// SIMATIC S7-200 SMART project (STEP 7-Micro/WIN SMART), CPU ST20

SYMBOL_TABLE System Symbols
Always_On        SM0.0    // Always ON
First_Scan_On    SM0.1    // ON for the first scan cycle only
Clock_1s         SM0.5    // Clock pulse that is ON for 0.5 s, OFF for 0.5 s, for a duty cycle time of 1 s.
END_SYMBOL_TABLE

SYMBOL_TABLE Modbus RTU Master2 (v2.0)
mModbusBufrFctn  VB420    // Modbusbufr[2] - function code byte
END_SYMBOL_TABLE

ORGANIZATION_BLOCK MAIN:OB1
TITLE=Program Comments
BEGIN
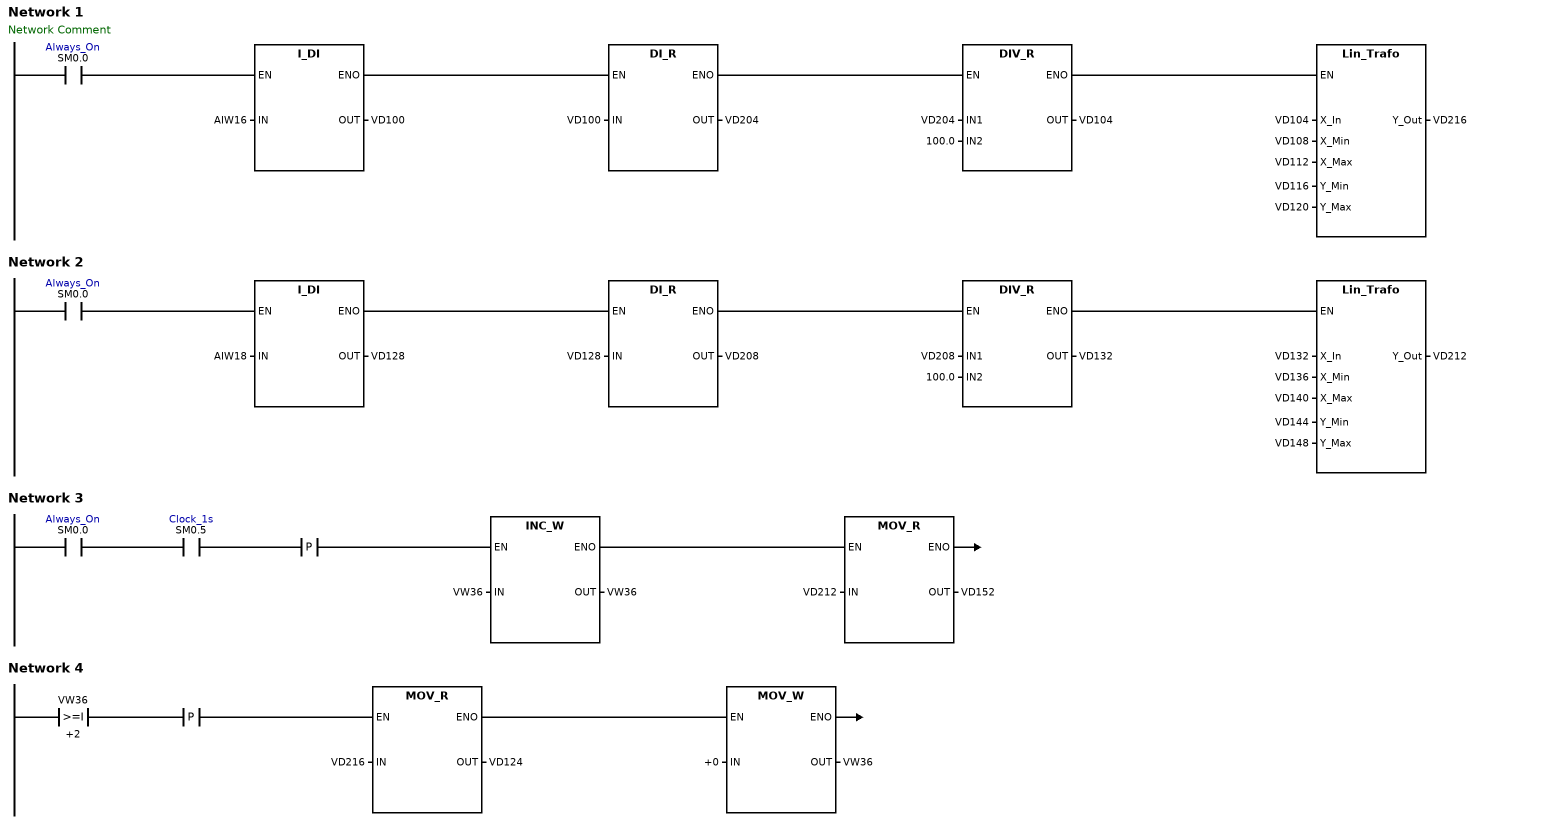
Network 1
// Network Comment
LD     Always_On:SM0.0
ITD    AIW16, VD100
AENO
DTR    VD100, VD204
AENO
MOVR   VD204, VD104
AENO
/R     100.0, VD104
AENO
CALL   Lin_Trafo:SBR1, VD104, VD108, VD112, VD116, VD120, VD216
Network 2
LD     Always_On:SM0.0
ITD    AIW18, VD128
AENO
DTR    VD128, VD208
AENO
MOVR   VD208, VD132
AENO
/R     100.0, VD132
AENO
CALL   Lin_Trafo:SBR1, VD132, VD136, VD140, VD144, VD148, VD212
Network 3
LD     Always_On:SM0.0
A      Clock_1s:SM0.5
EU
INCW   VW36
AENO
MOVR   VD212, VD152
Network 4
LDW>=  VW36, +2
EU
MOVR   VD216, VD124
AENO
MOVW   +0, VW36
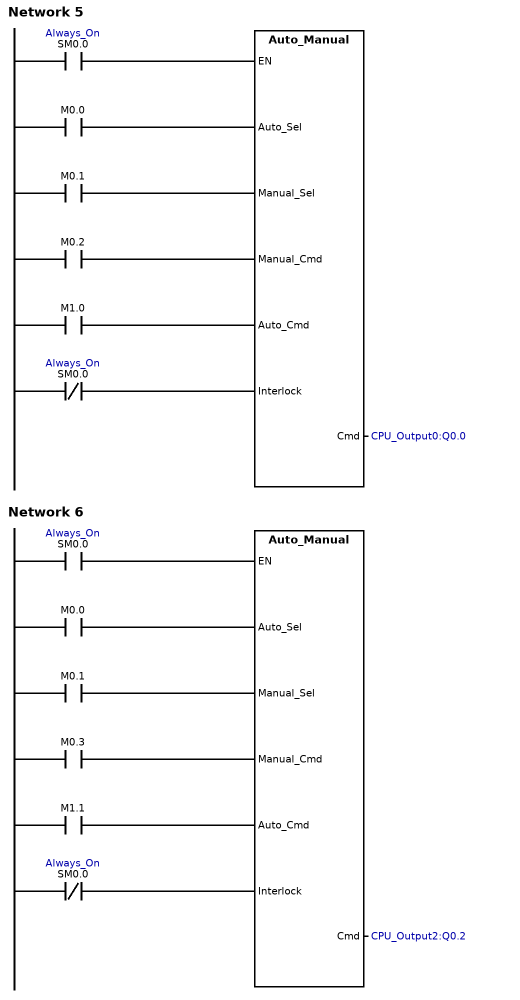
Network 5
LD     Always_On:SM0.0
=      L60.0
LD     M0.0
=      L63.7
LD     M0.1
=      L63.6
LD     M0.2
=      L63.5
LD     M1.0
=      L63.4
LDN    Always_On:SM0.0
=      L63.3
LD     L60.0
CALL   Auto_Manual:SBR2, L63.7, L63.6, L63.5, L63.4, L63.3, CPU_Output0:Q0.0
Network 6
LD     Always_On:SM0.0
=      L60.0
LD     M0.0
=      L63.7
LD     M0.1
=      L63.6
LD     M0.3
=      L63.5
LD     M1.1
=      L63.4
LDN    Always_On:SM0.0
=      L63.3
LD     L60.0
CALL   Auto_Manual:SBR2, L63.7, L63.6, L63.5, L63.4, L63.3, CPU_Output2:Q0.2
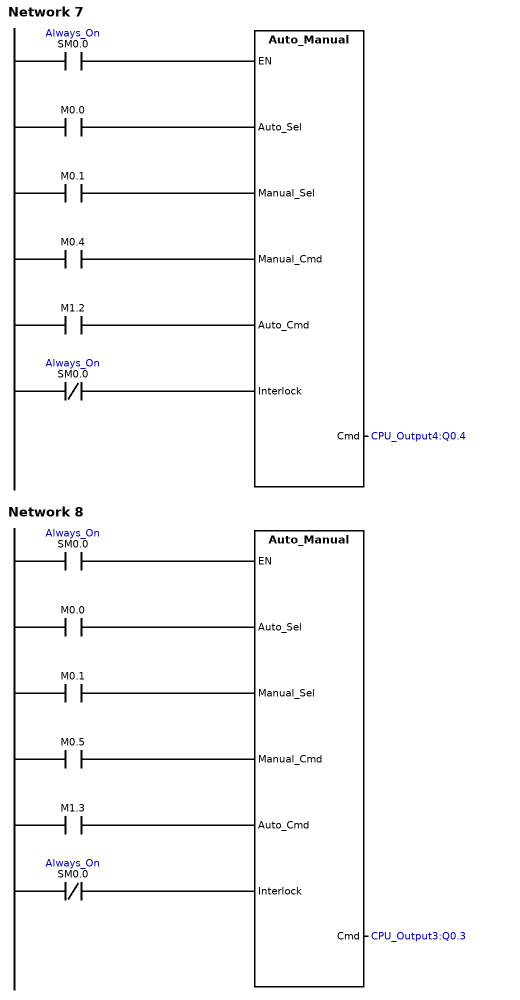
Network 7
LD     Always_On:SM0.0
=      L60.0
LD     M0.0
=      L63.7
LD     M0.1
=      L63.6
LD     M0.4
=      L63.5
LD     M1.2
=      L63.4
LDN    Always_On:SM0.0
=      L63.3
LD     L60.0
CALL   Auto_Manual:SBR2, L63.7, L63.6, L63.5, L63.4, L63.3, CPU_Output4:Q0.4
Network 8
LD     Always_On:SM0.0
=      L60.0
LD     M0.0
=      L63.7
LD     M0.1
=      L63.6
LD     M0.5
=      L63.5
LD     M1.3
=      L63.4
LDN    Always_On:SM0.0
=      L63.3
LD     L60.0
CALL   Auto_Manual:SBR2, L63.7, L63.6, L63.5, L63.4, L63.3, CPU_Output3:Q0.3
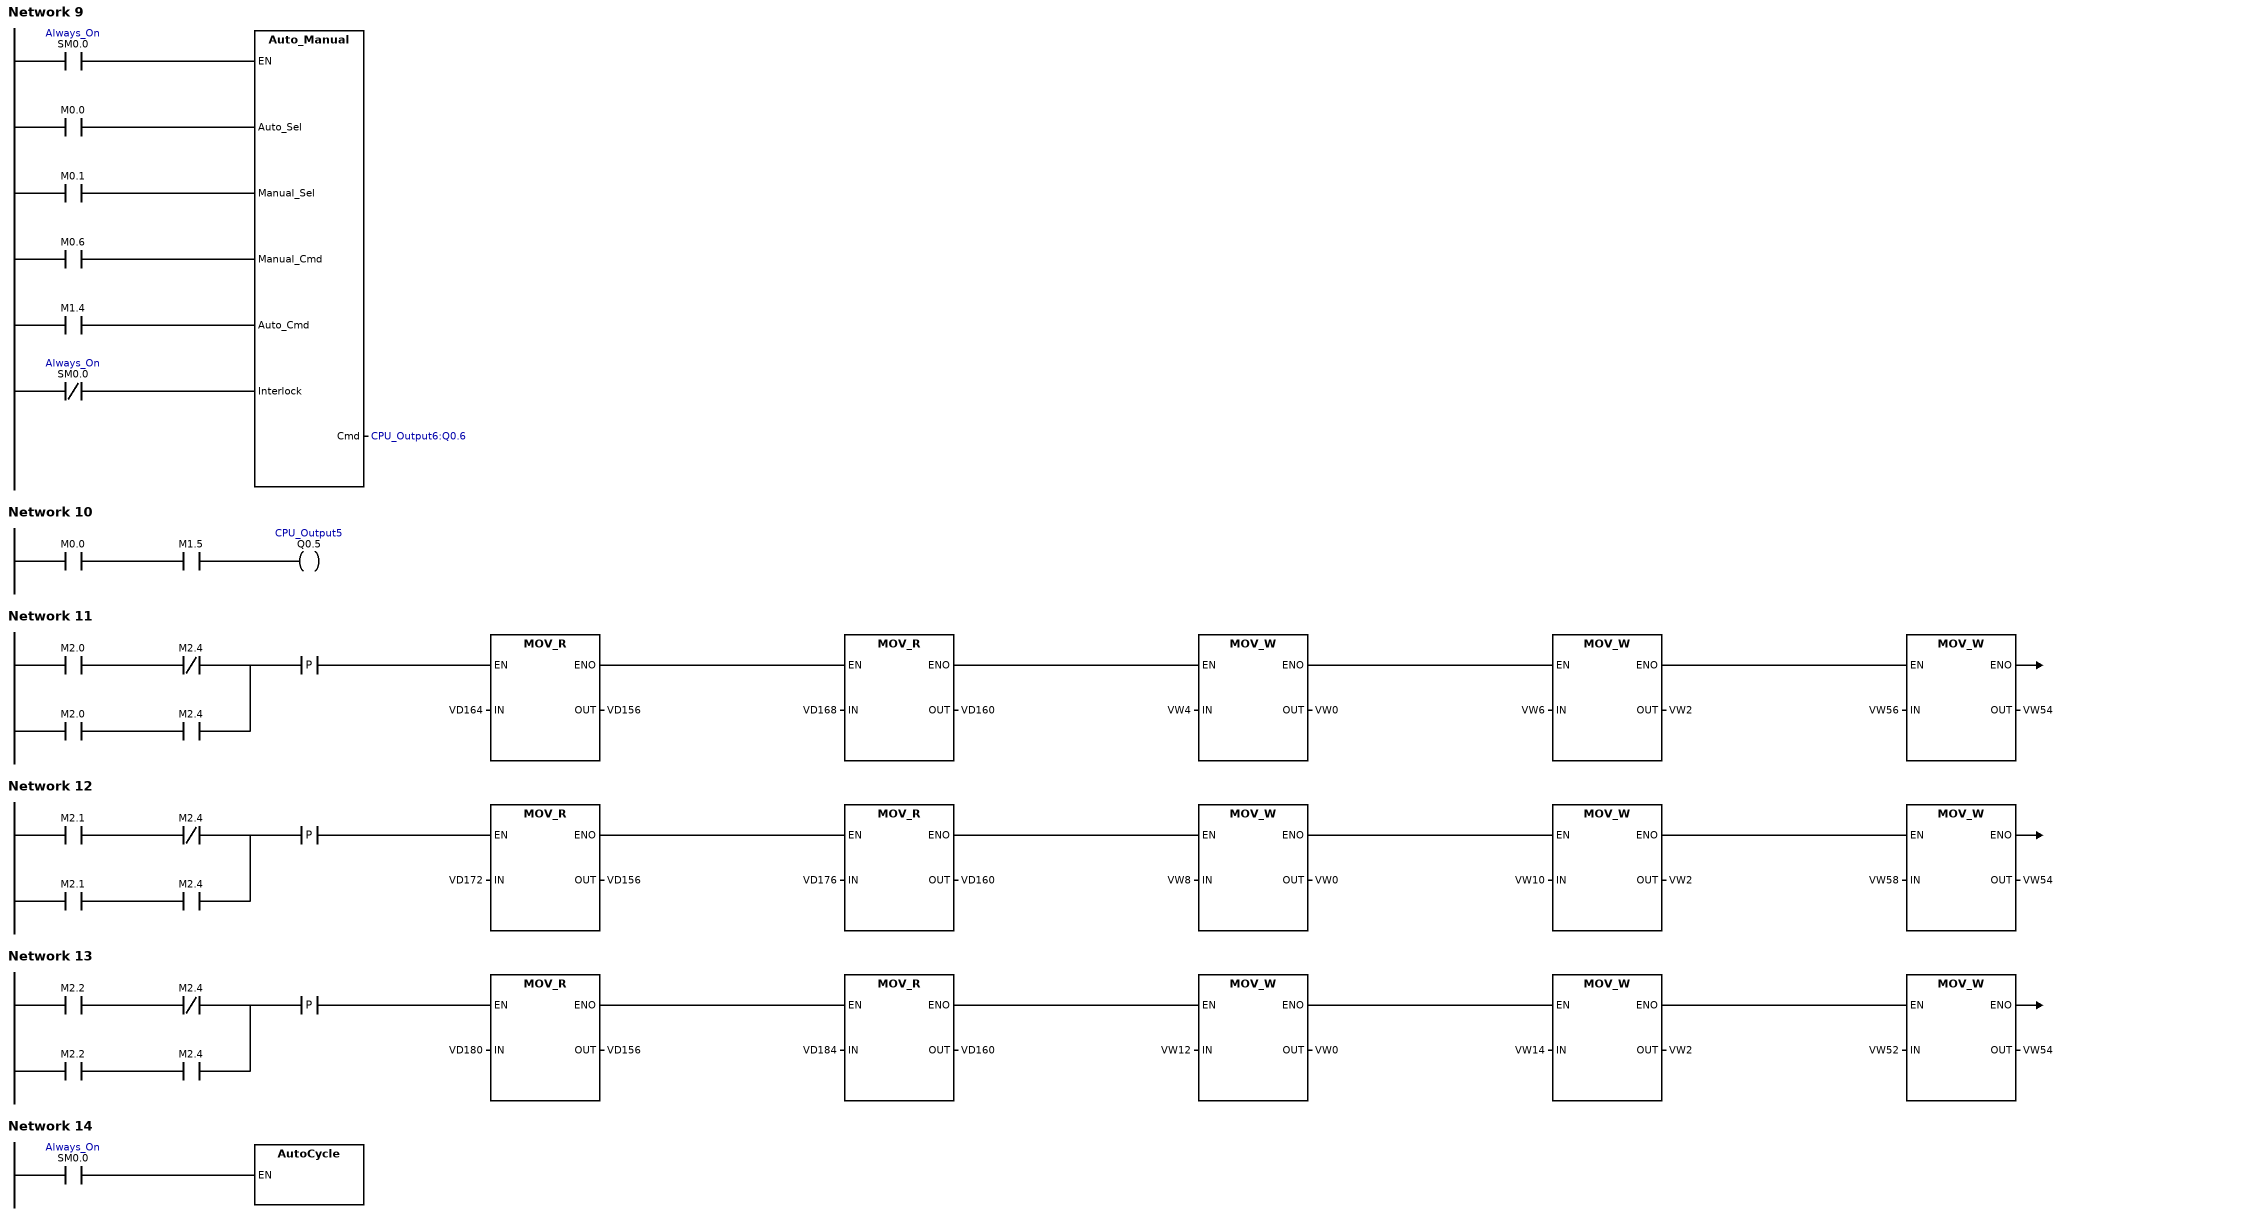
Network 9
LD     Always_On:SM0.0
=      L60.0
LD     M0.0
=      L63.7
LD     M0.1
=      L63.6
LD     M0.6
=      L63.5
LD     M1.4
=      L63.4
LDN    Always_On:SM0.0
=      L63.3
LD     L60.0
CALL   Auto_Manual:SBR2, L63.7, L63.6, L63.5, L63.4, L63.3, CPU_Output6:Q0.6
Network 10
LD     M0.0
A      M1.5
=      CPU_Output5:Q0.5
Network 11
LD     M2.0
AN     M2.4
LD     M2.0
A      M2.4
OLD
EU
MOVR   VD164, VD156
AENO
MOVR   VD168, VD160
AENO
MOVW   VW4, VW0
AENO
MOVW   VW6, VW2
AENO
MOVW   VW56, VW54
Network 12
LD     M2.1
AN     M2.4
LD     M2.1
A      M2.4
OLD
EU
MOVR   VD172, VD156
AENO
MOVR   VD176, VD160
AENO
MOVW   VW8, VW0
AENO
MOVW   VW10, VW2
AENO
MOVW   VW58, VW54
Network 13
LD     M2.2
AN     M2.4
LD     M2.2
A      M2.4
OLD
EU
MOVR   VD180, VD156
AENO
MOVR   VD184, VD160
AENO
MOVW   VW12, VW0
AENO
MOVW   VW14, VW2
AENO
MOVW   VW52, VW54
Network 14
LD     Always_On:SM0.0
CALL   AutoCycle:SBR0
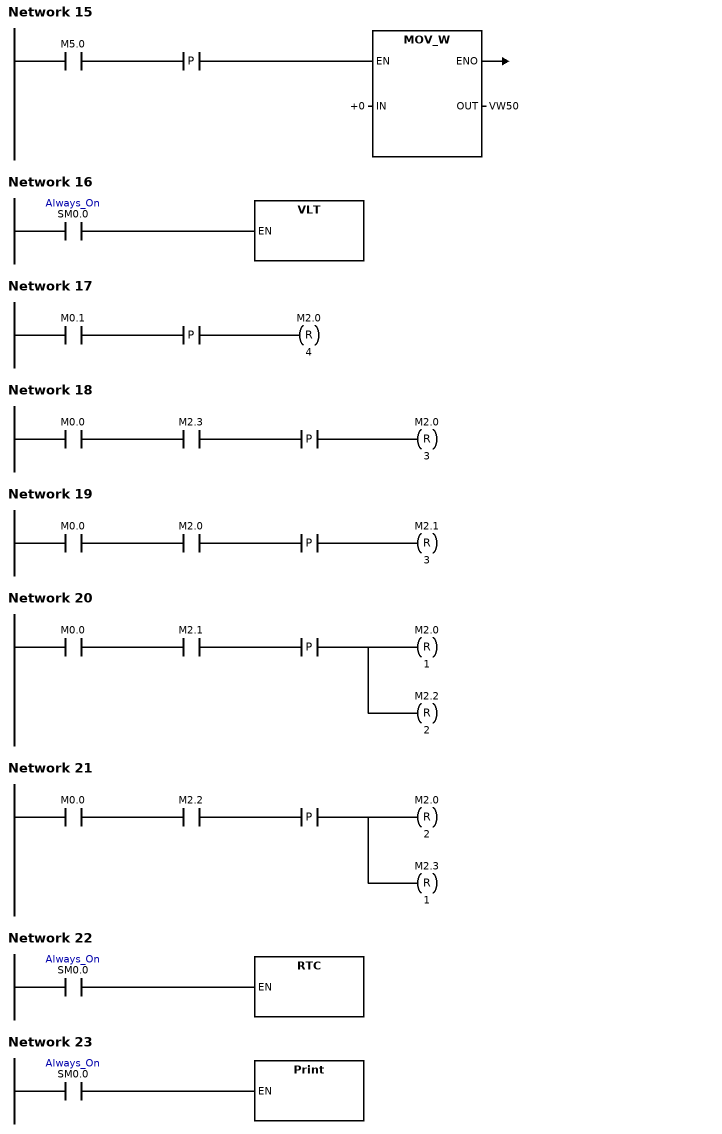
Network 15
LD     M5.0
EU
MOVW   +0, VW50
Network 16
LD     Always_On:SM0.0
CALL   VLT:SBR5
Network 17
LD     M0.1
EU
R      M2.0, 4
Network 18
LD     M0.0
A      M2.3
EU
R      M2.0, 3
Network 19
LD     M0.0
A      M2.0
EU
R      M2.1, 3
Network 20
LD     M0.0
A      M2.1
EU
R      M2.0, 1
R      M2.2, 2
Network 21
LD     M0.0
A      M2.2
EU
R      M2.0, 2
R      M2.3, 1
Network 22
LD     Always_On:SM0.0
CALL   RTC:SBR7
Network 23
LD     Always_On:SM0.0
CALL   Print:SBR8
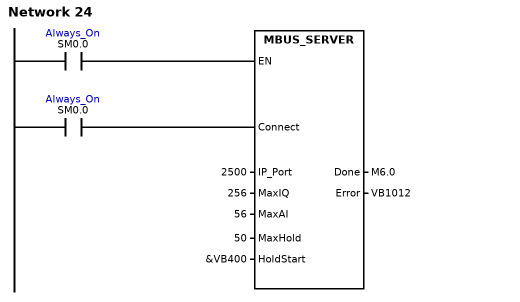
Network 24
LD     Always_On:SM0.0
=      L60.0
LD     Always_On:SM0.0
=      L63.7
LD     L60.0
CALL   MBUS_SERVER:SBR6, L63.7, 2500, 256, 56, 50, &VB400, M6.0, VB1012
END_ORGANIZATION_BLOCK

SUBROUTINE_BLOCK AutoCycle:SBR0
TITLE=Subroutine Comments
BEGIN
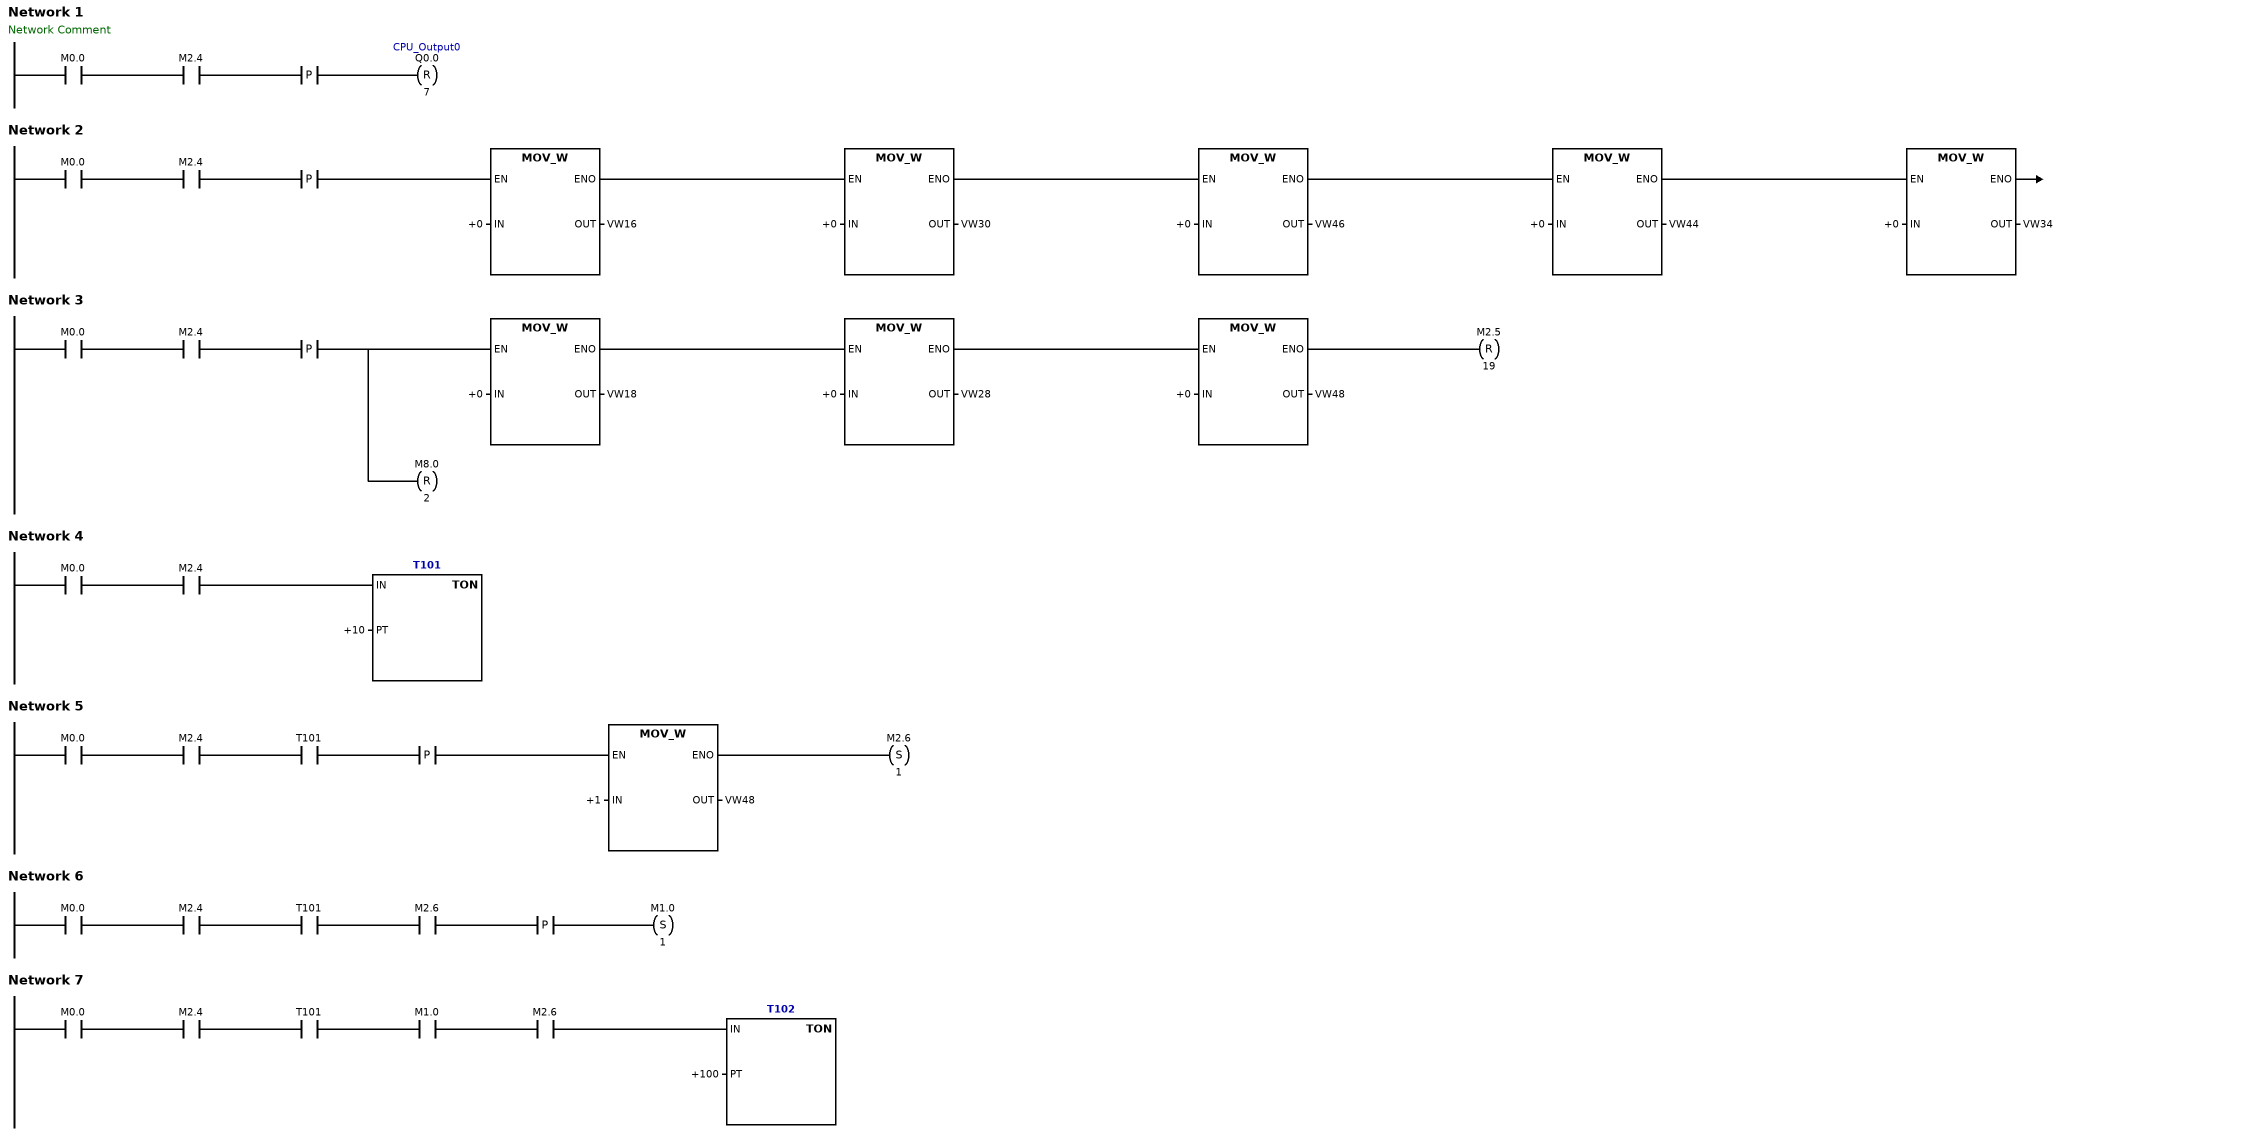
Network 1
// Network Comment
LD     M0.0
A      M2.4
EU
R      CPU_Output0:Q0.0, 7
Network 2
LD     M0.0
A      M2.4
EU
MOVW   +0, VW16
AENO
MOVW   +0, VW30
AENO
MOVW   +0, VW46
AENO
MOVW   +0, VW44
AENO
MOVW   +0, VW34
Network 3
LD     M0.0
A      M2.4
EU
LPS
MOVW   +0, VW18
AENO
MOVW   +0, VW28
AENO
MOVW   +0, VW48
AENO
R      M2.5, 19
LPP
R      M8.0, 2
Network 4
LD     M0.0
A      M2.4
TON    T101, +10
Network 5
LD     M0.0
A      M2.4
A      T101
EU
MOVW   +1, VW48
AENO
S      M2.6, 1
Network 6
LD     M0.0
A      M2.4
A      T101
A      M2.6
EU
S      M1.0, 1
Network 7
LD     M0.0
A      M2.4
A      T101
A      M1.0
A      M2.6
TON    T102, +100
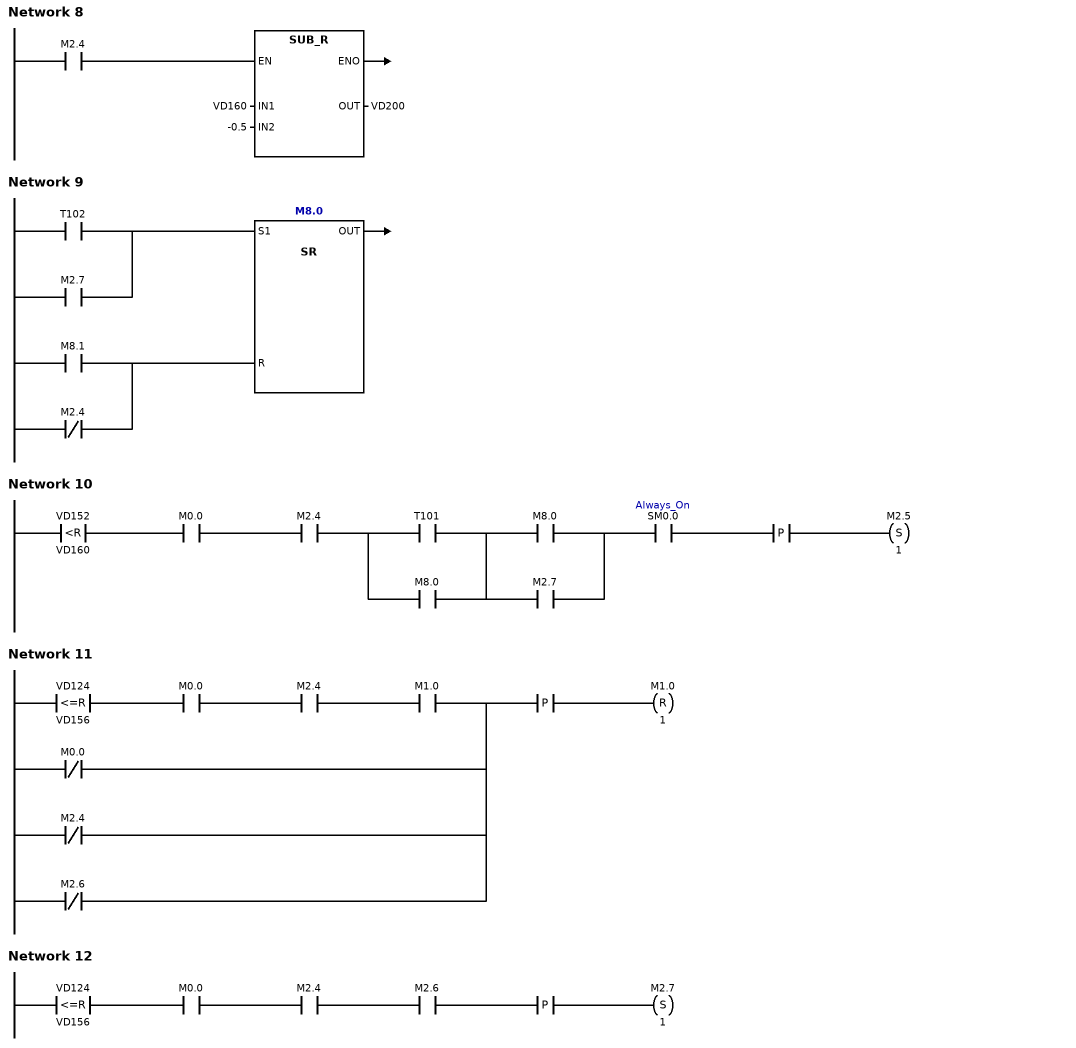
Network 8
LD     M2.4
MOVR   VD160, VD200
-R     -0.5, VD200
Network 9
LD     T102
O      M2.7
LD     M8.1
ON     M2.4
NOT
A      M8.0
OLD
=      M8.0
Network 10
LDR<   VD152, VD160
A      M0.0
A      M2.4
LD     T101
O      M8.0
ALD
LD     M8.0
O      M2.7
ALD
A      Always_On:SM0.0
EU
S      M2.5, 1
Network 11
LDR<=  VD124, VD156
A      M0.0
A      M2.4
A      M1.0
ON     M0.0
ON     M2.4
ON     M2.6
EU
R      M1.0, 1
Network 12
LDR<=  VD124, VD156
A      M0.0
A      M2.4
A      M2.6
EU
S      M2.7, 1
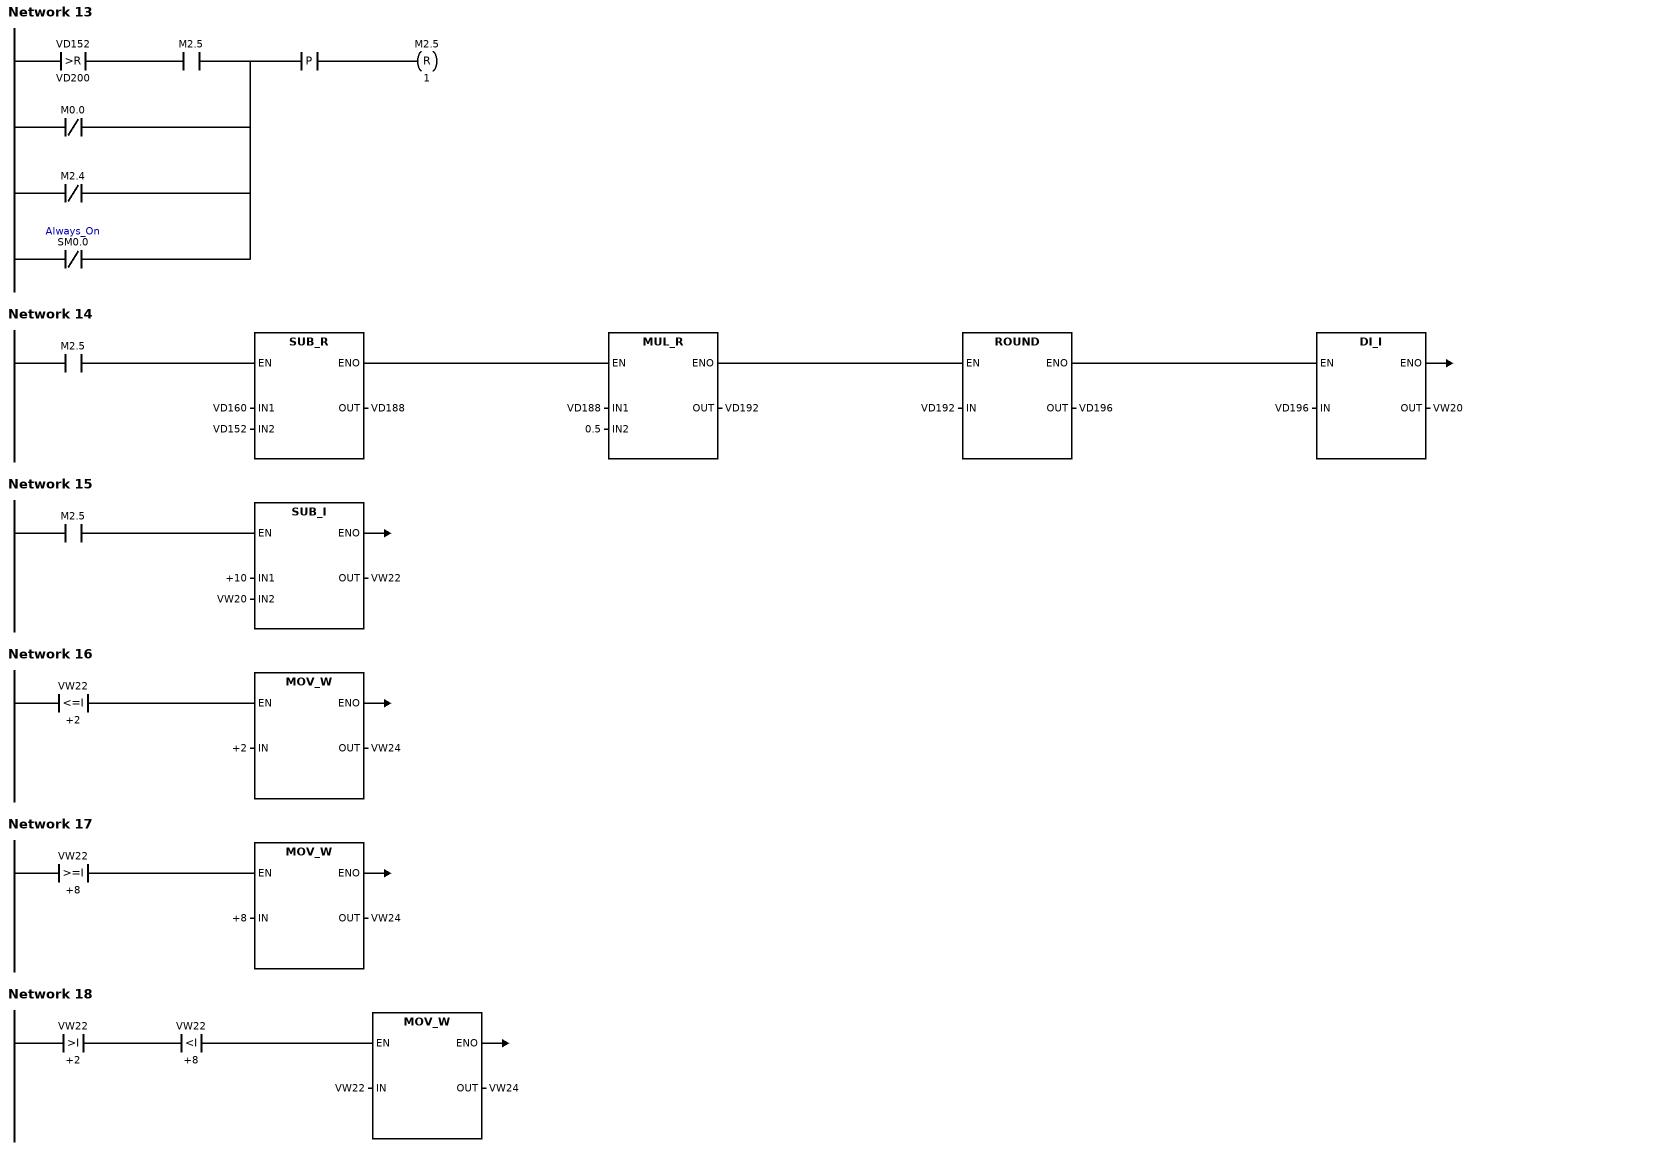
Network 13
LDR>   VD152, VD200
A      M2.5
ON     M0.0
ON     M2.4
ON     Always_On:SM0.0
EU
R      M2.5, 1
Network 14
LD     M2.5
MOVR   VD160, VD188
AENO
-R     VD152, VD188
AENO
MOVR   VD188, VD192
AENO
*R     0.5, VD192
AENO
ROUND  VD192, VD196
AENO
DTI    VD196, VW20
Network 15
LD     M2.5
MOVW   +10, VW22
-I     VW20, VW22
Network 16
LDW<=  VW22, +2
MOVW   +2, VW24
Network 17
LDW>=  VW22, +8
MOVW   +8, VW24
Network 18
LDW>   VW22, +2
AW<    VW22, +8
MOVW   VW22, VW24
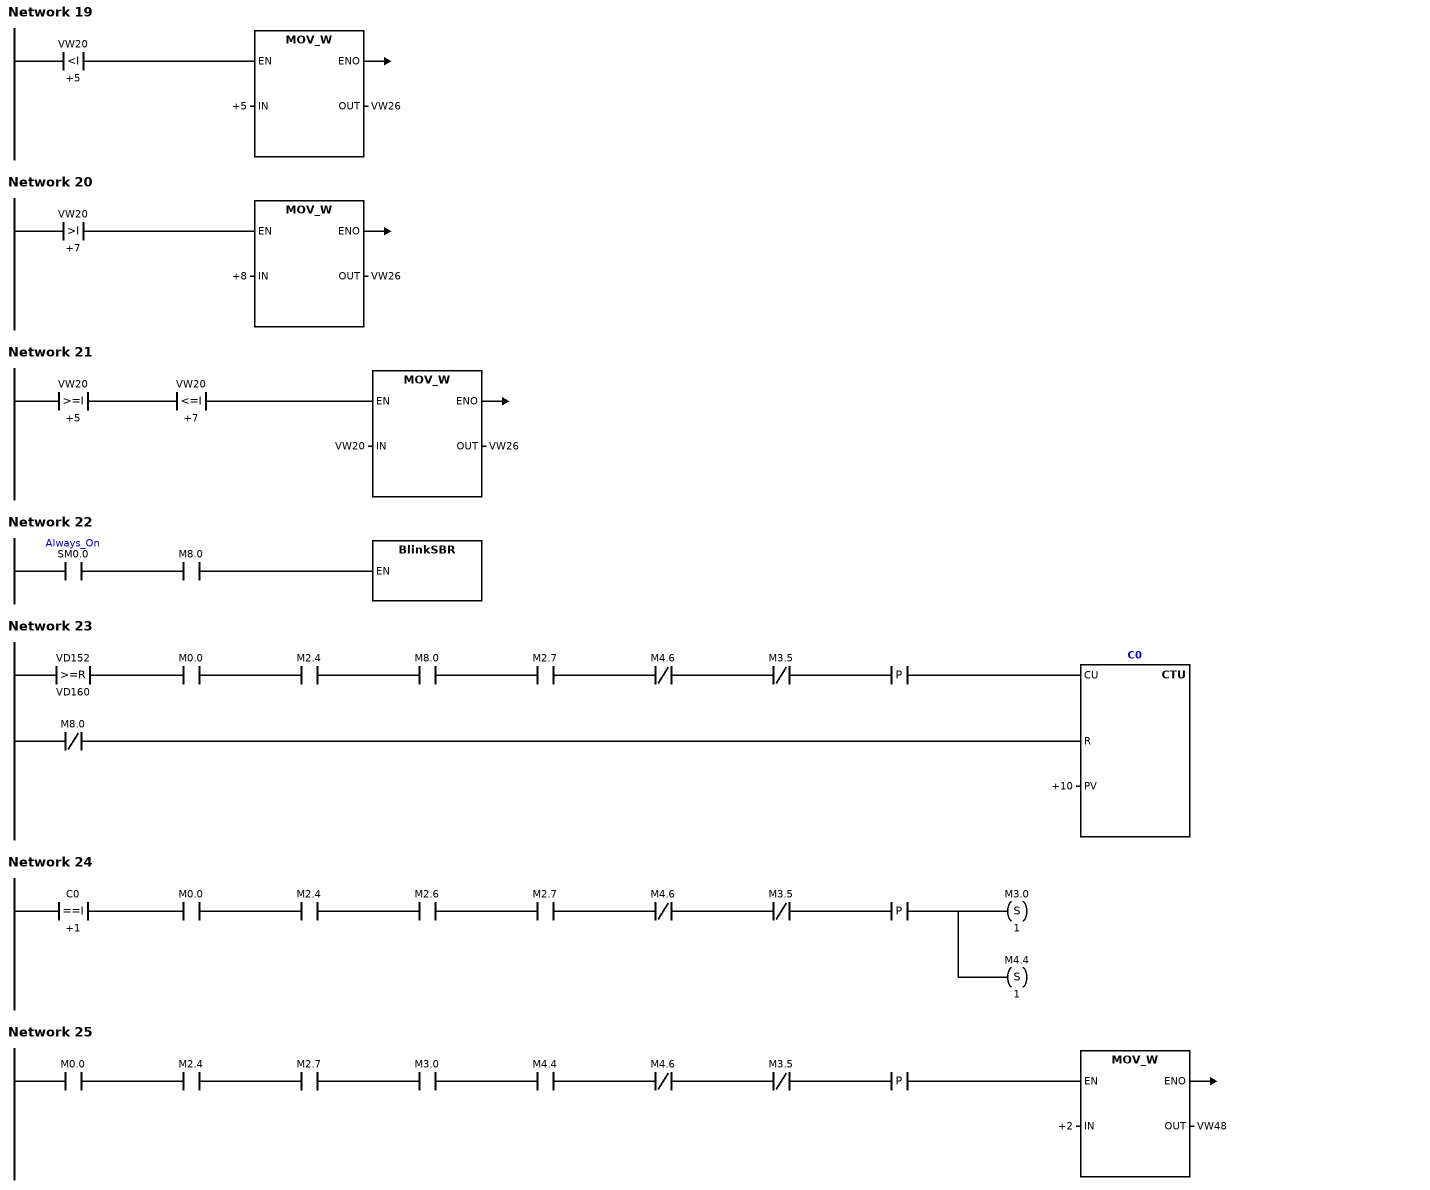
Network 19
LDW<   VW20, +5
MOVW   +5, VW26
Network 20
LDW>   VW20, +7
MOVW   +8, VW26
Network 21
LDW>=  VW20, +5
AW<=   VW20, +7
MOVW   VW20, VW26
Network 22
LD     Always_On:SM0.0
A      M8.0
CALL   BlinkSBR:SBR4
Network 23
LDR>=  VD152, VD160
A      M0.0
A      M2.4
A      M8.0
A      M2.7
AN     M4.6
AN     M3.5
EU
LDN    M8.0
CTU    C0, +10
Network 24
LDW=   C0, +1
A      M0.0
A      M2.4
A      M2.6
A      M2.7
AN     M4.6
AN     M3.5
EU
S      M3.0, 1
S      M4.4, 1
Network 25
LD     M0.0
A      M2.4
A      M2.7
A      M3.0
A      M4.4
AN     M4.6
AN     M3.5
EU
MOVW   +2, VW48
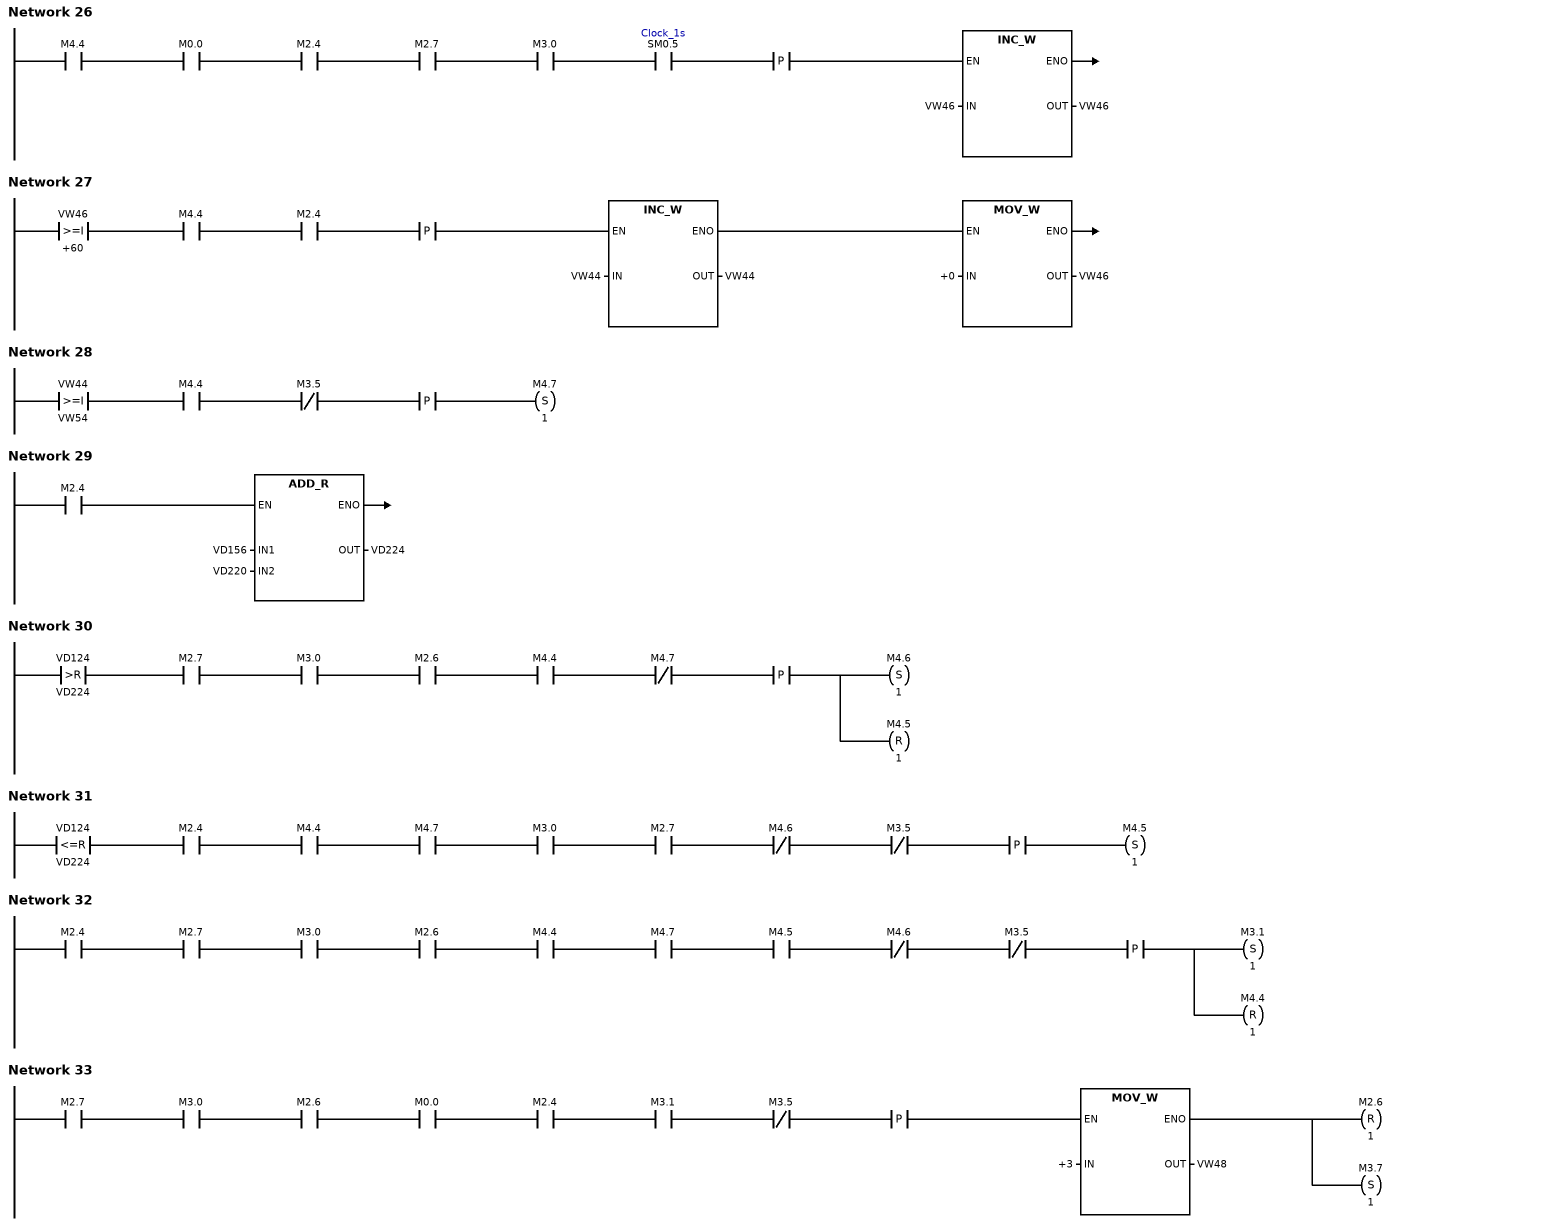
Network 26
LD     M4.4
A      M0.0
A      M2.4
A      M2.7
A      M3.0
A      Clock_1s:SM0.5
EU
INCW   VW46
Network 27
LDW>=  VW46, +60
A      M4.4
A      M2.4
EU
INCW   VW44
AENO
MOVW   +0, VW46
Network 28
LDW>=  VW44, VW54
A      M4.4
AN     M3.5
EU
S      M4.7, 1
Network 29
LD     M2.4
MOVR   VD156, VD224
+R     VD220, VD224
Network 30
LDR>   VD124, VD224
A      M2.7
A      M3.0
A      M2.6
A      M4.4
AN     M4.7
EU
S      M4.6, 1
R      M4.5, 1
Network 31
LDR<=  VD124, VD224
A      M2.4
A      M4.4
A      M4.7
A      M3.0
A      M2.7
AN     M4.6
AN     M3.5
EU
S      M4.5, 1
Network 32
LD     M2.4
A      M2.7
A      M3.0
A      M2.6
A      M4.4
A      M4.7
A      M4.5
AN     M4.6
AN     M3.5
EU
S      M3.1, 1
R      M4.4, 1
Network 33
LD     M2.7
A      M3.0
A      M2.6
A      M0.0
A      M2.4
A      M3.1
AN     M3.5
EU
MOVW   +3, VW48
AENO
R      M2.6, 1
S      M3.7, 1
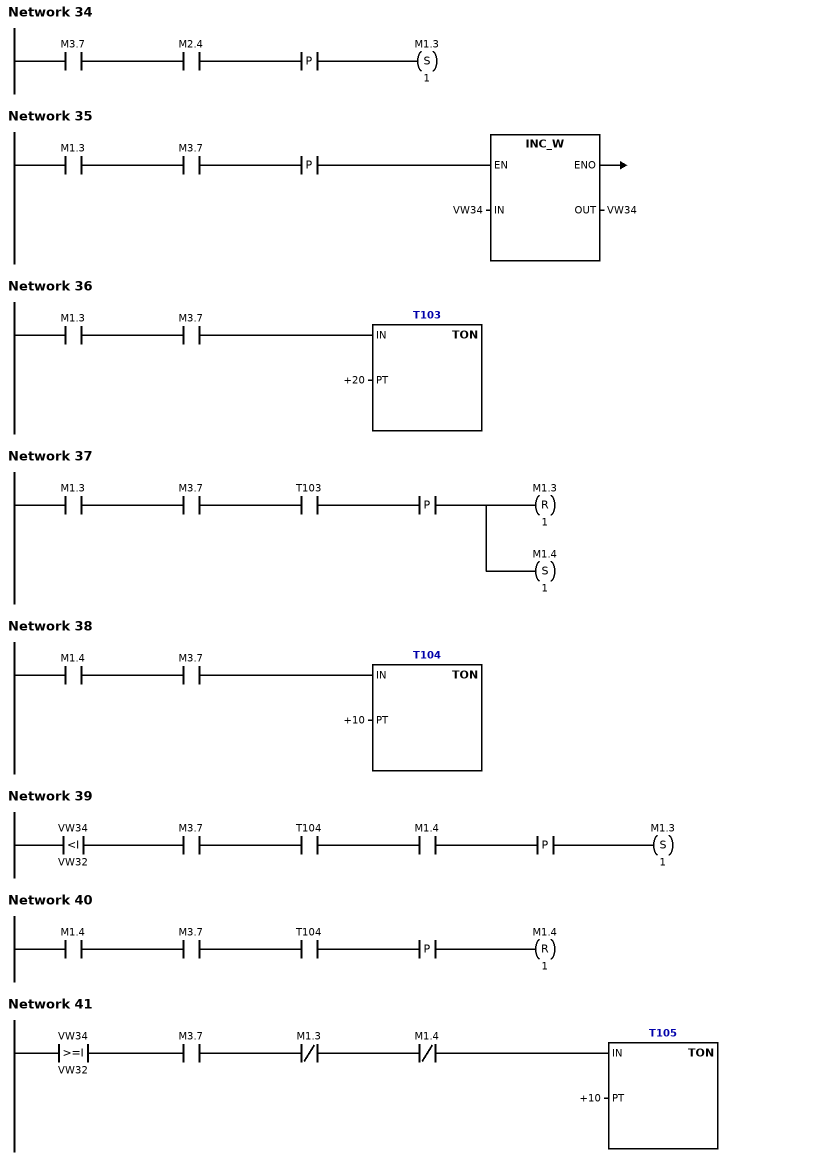
Network 34
LD     M3.7
A      M2.4
EU
S      M1.3, 1
Network 35
LD     M1.3
A      M3.7
EU
INCW   VW34
Network 36
LD     M1.3
A      M3.7
TON    T103, +20
Network 37
LD     M1.3
A      M3.7
A      T103
EU
R      M1.3, 1
S      M1.4, 1
Network 38
LD     M1.4
A      M3.7
TON    T104, +10
Network 39
LDW<   VW34, VW32
A      M3.7
A      T104
A      M1.4
EU
S      M1.3, 1
Network 40
LD     M1.4
A      M3.7
A      T104
EU
R      M1.4, 1
Network 41
LDW>=  VW34, VW32
A      M3.7
AN     M1.3
AN     M1.4
TON    T105, +10
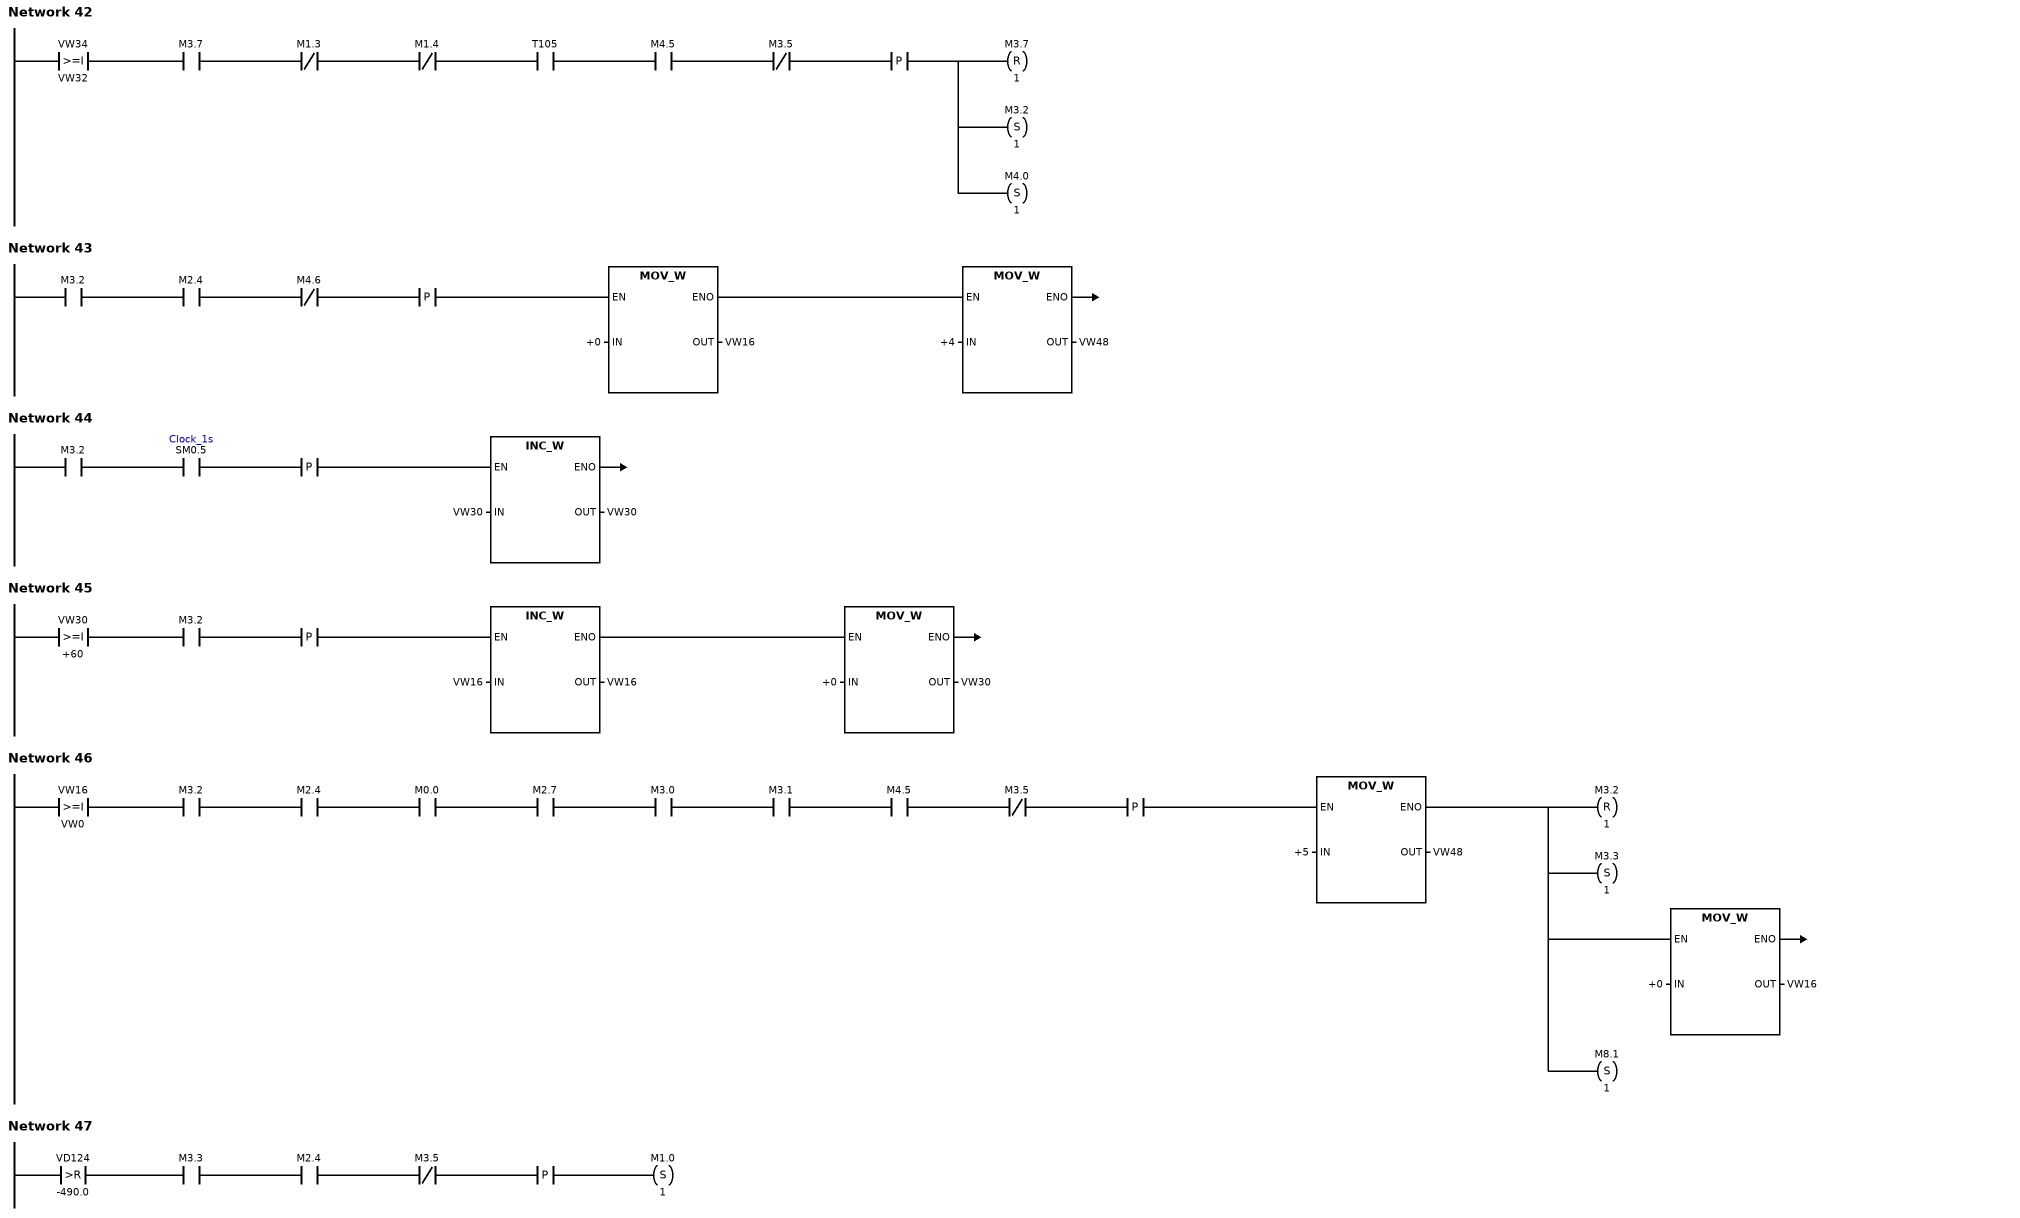
Network 42
LDW>=  VW34, VW32
A      M3.7
AN     M1.3
AN     M1.4
A      T105
A      M4.5
AN     M3.5
EU
R      M3.7, 1
S      M3.2, 1
S      M4.0, 1
Network 43
LD     M3.2
A      M2.4
AN     M4.6
EU
MOVW   +0, VW16
AENO
MOVW   +4, VW48
Network 44
LD     M3.2
A      Clock_1s:SM0.5
EU
INCW   VW30
Network 45
LDW>=  VW30, +60
A      M3.2
EU
INCW   VW16
AENO
MOVW   +0, VW30
Network 46
LDW>=  VW16, VW0
A      M3.2
A      M2.4
A      M0.0
A      M2.7
A      M3.0
A      M3.1
A      M4.5
AN     M3.5
EU
MOVW   +5, VW48
AENO
R      M3.2, 1
S      M3.3, 1
MOVW   +0, VW16
S      M8.1, 1
Network 47
LDR>   VD124, -490.0
A      M3.3
A      M2.4
AN     M3.5
EU
S      M1.0, 1
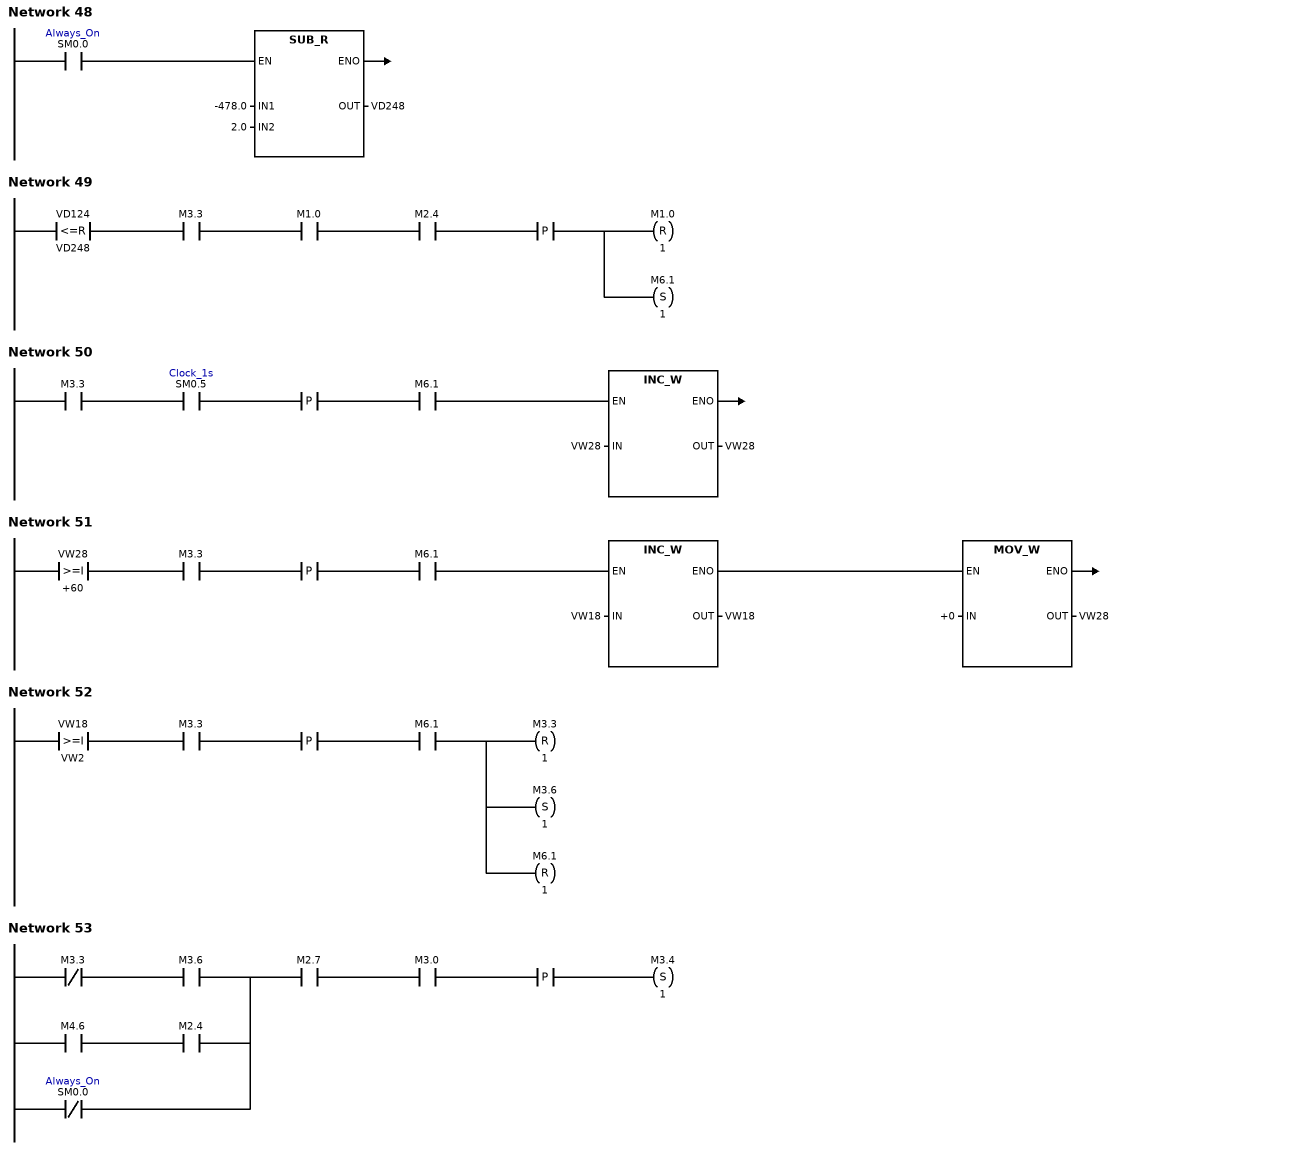
Network 48
LD     Always_On:SM0.0
MOVR   -478.0, VD248
-R     2.0, VD248
Network 49
LDR<=  VD124, VD248
A      M3.3
A      M1.0
A      M2.4
EU
R      M1.0, 1
S      M6.1, 1
Network 50
LD     M3.3
A      Clock_1s:SM0.5
EU
A      M6.1
INCW   VW28
Network 51
LDW>=  VW28, +60
A      M3.3
EU
A      M6.1
INCW   VW18
AENO
MOVW   +0, VW28
Network 52
LDW>=  VW18, VW2
A      M3.3
EU
A      M6.1
R      M3.3, 1
S      M3.6, 1
R      M6.1, 1
Network 53
LDN    M3.3
A      M3.6
LD     M4.6
A      M2.4
OLD
ON     Always_On:SM0.0
A      M2.7
A      M3.0
EU
S      M3.4, 1
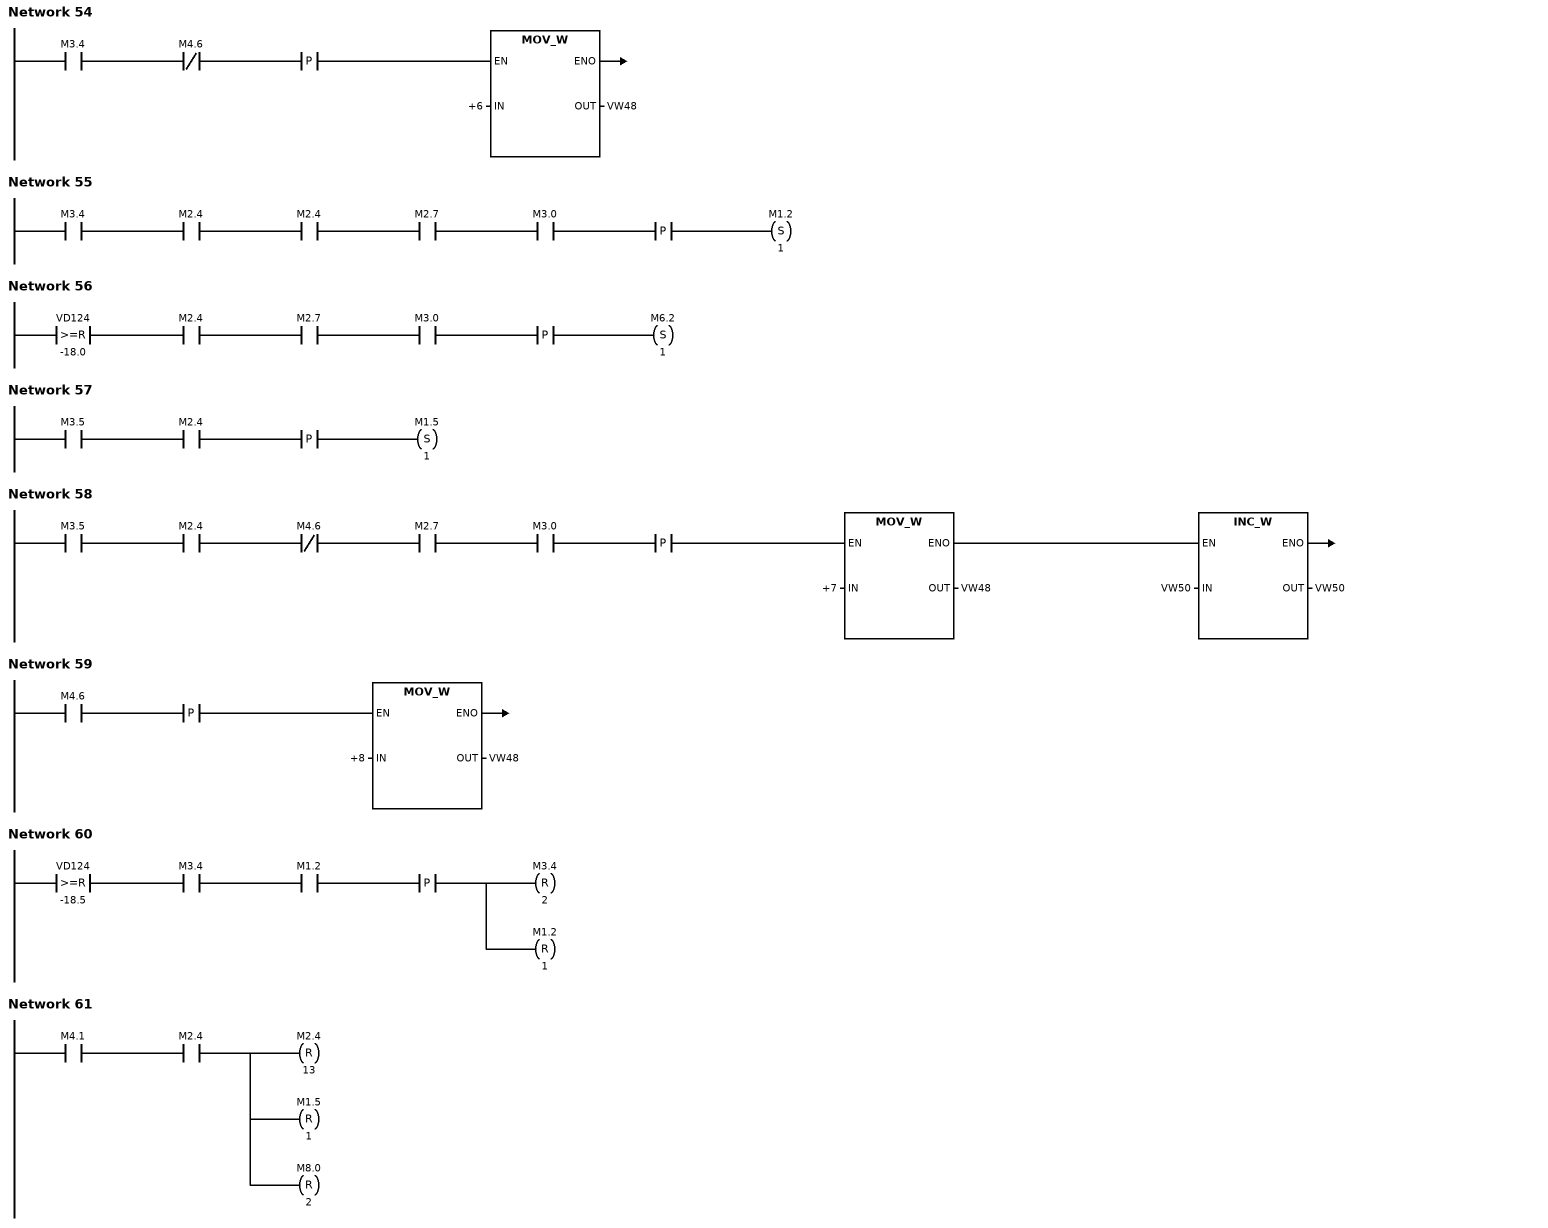
Network 54
LD     M3.4
AN     M4.6
EU
MOVW   +6, VW48
Network 55
LD     M3.4
A      M2.4
A      M2.4
A      M2.7
A      M3.0
EU
S      M1.2, 1
Network 56
LDR>=  VD124, -18.0
A      M2.4
A      M2.7
A      M3.0
EU
S      M6.2, 1
Network 57
LD     M3.5
A      M2.4
EU
S      M1.5, 1
Network 58
LD     M3.5
A      M2.4
AN     M4.6
A      M2.7
A      M3.0
EU
MOVW   +7, VW48
AENO
INCW   VW50
Network 59
LD     M4.6
EU
MOVW   +8, VW48
Network 60
LDR>=  VD124, -18.5
A      M3.4
A      M1.2
EU
R      M3.4, 2
R      M1.2, 1
Network 61
LD     M4.1
A      M2.4
R      M2.4, 13
R      M1.5, 1
R      M8.0, 2
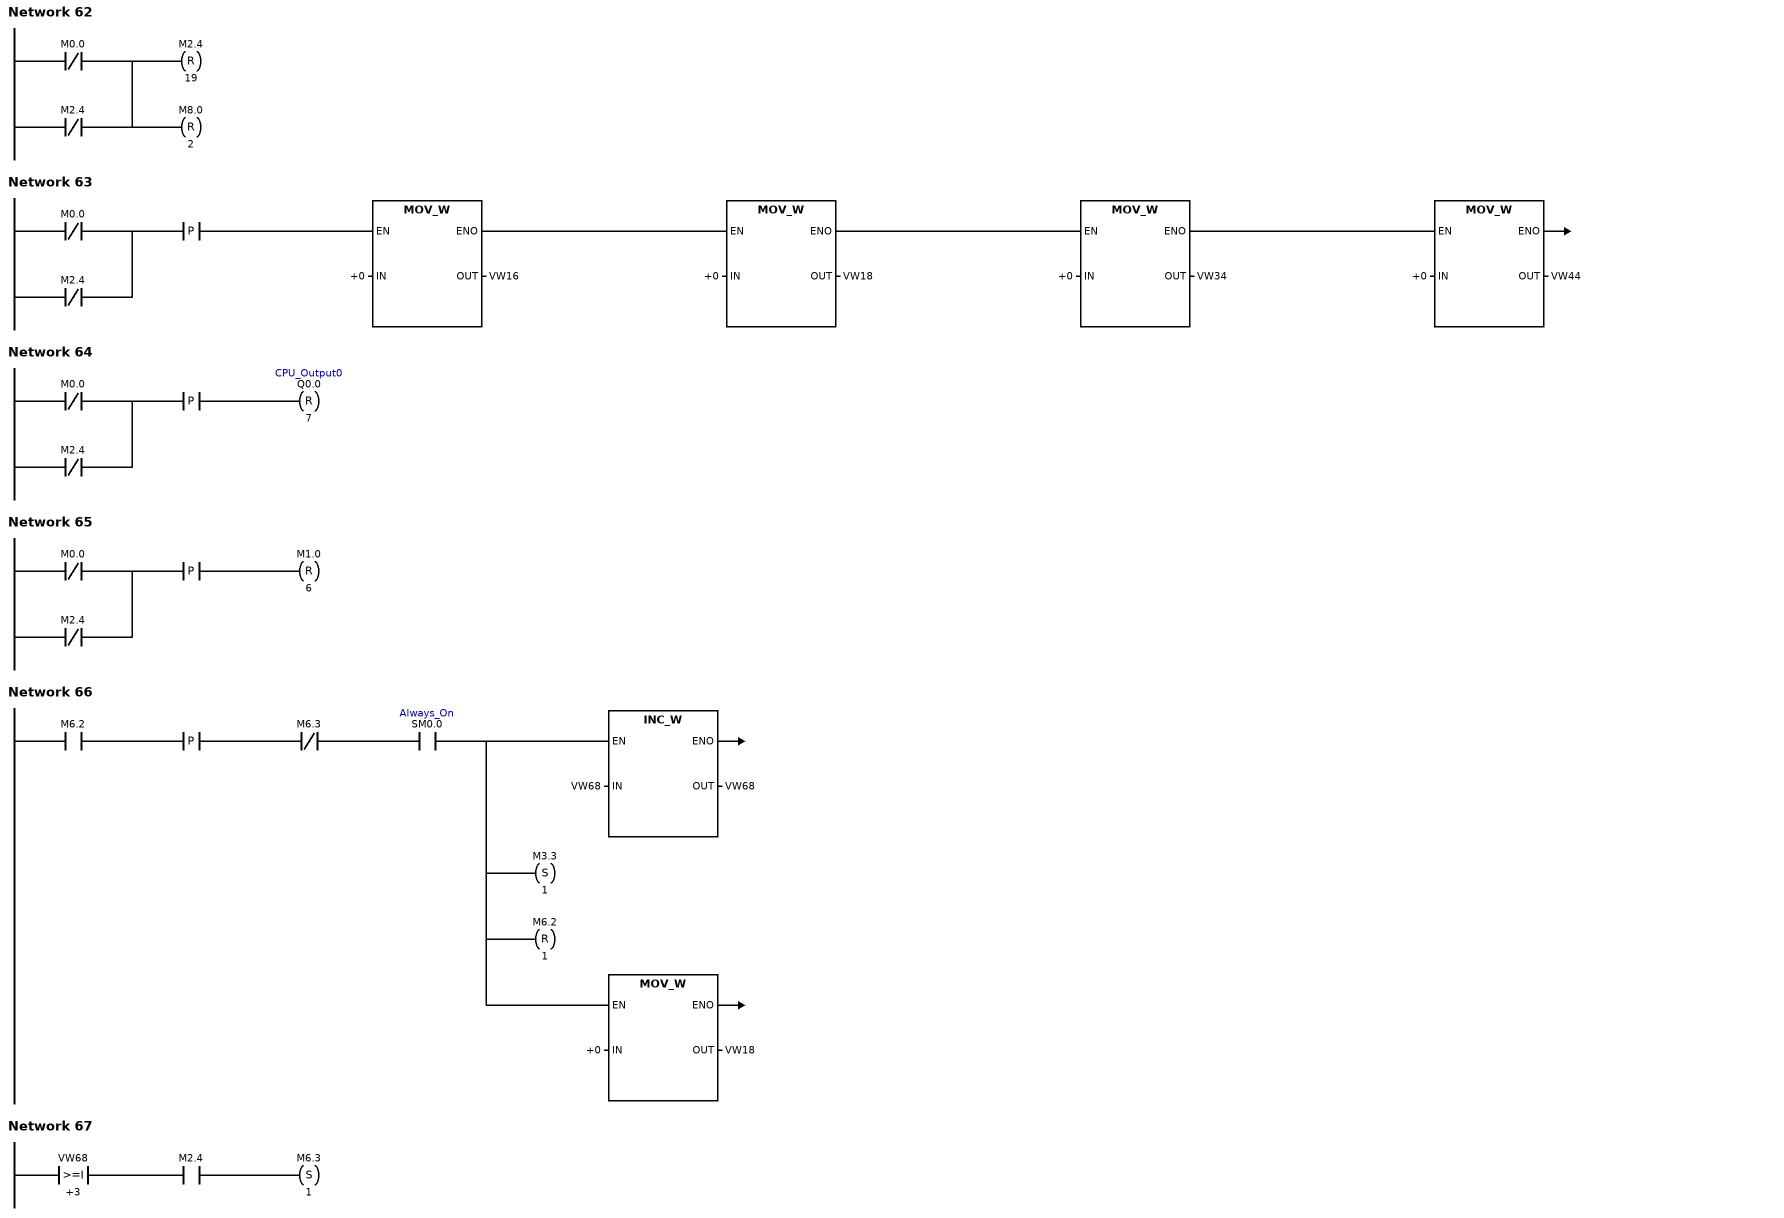
Network 62
LDN    M0.0
ON     M2.4
R      M2.4, 19
R      M8.0, 2
Network 63
LDN    M0.0
ON     M2.4
EU
MOVW   +0, VW16
AENO
MOVW   +0, VW18
AENO
MOVW   +0, VW34
AENO
MOVW   +0, VW44
Network 64
LDN    M0.0
ON     M2.4
EU
R      CPU_Output0:Q0.0, 7
Network 65
LDN    M0.0
ON     M2.4
EU
R      M1.0, 6
Network 66
LD     M6.2
EU
AN     M6.3
A      Always_On:SM0.0
INCW   VW68
S      M3.3, 1
R      M6.2, 1
MOVW   +0, VW18
Network 67
LDW>=  VW68, +3
A      M2.4
S      M6.3, 1
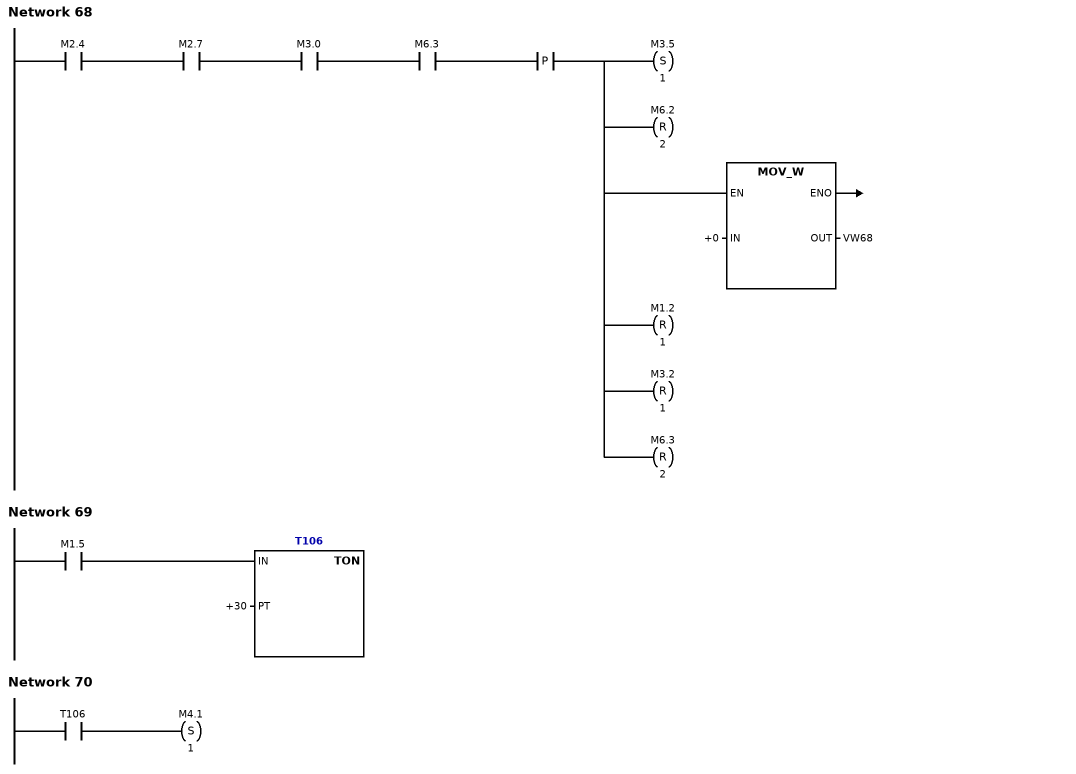
Network 68
LD     M2.4
A      M2.7
A      M3.0
A      M6.3
EU
S      M3.5, 1
R      M6.2, 2
MOVW   +0, VW68
R      M1.2, 1
R      M3.2, 1
R      M6.3, 2
Network 69
LD     M1.5
TON    T106, +30
Network 70
LD     T106
S      M4.1, 1
END_SUBROUTINE_BLOCK

// SBR1: protected block, not included

// SBR2: protected block, not included

// SBR3: protected block, not included

SUBROUTINE_BLOCK BlinkSBR:SBR4
TITLE=
BEGIN
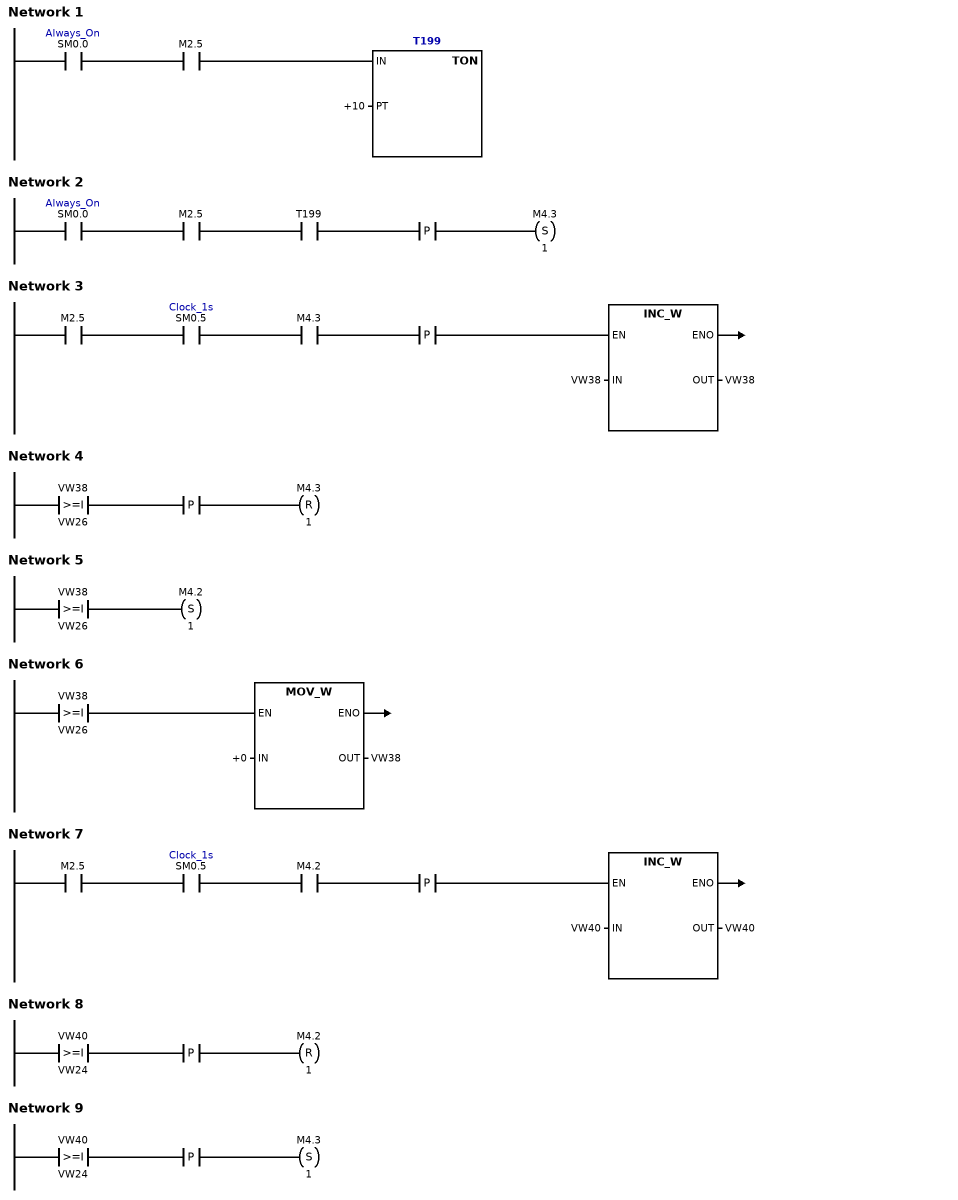
Network 1
LD     Always_On:SM0.0
A      M2.5
TON    T199, +10
Network 2
LD     Always_On:SM0.0
A      M2.5
A      T199
EU
S      M4.3, 1
Network 3
LD     M2.5
A      Clock_1s:SM0.5
A      M4.3
EU
INCW   VW38
Network 4
LDW>=  VW38, VW26
EU
R      M4.3, 1
Network 5
LDW>=  VW38, VW26
S      M4.2, 1
Network 6
LDW>=  VW38, VW26
MOVW   +0, VW38
Network 7
LD     M2.5
A      Clock_1s:SM0.5
A      M4.2
EU
INCW   VW40
Network 8
LDW>=  VW40, VW24
EU
R      M4.2, 1
Network 9
LDW>=  VW40, VW24
EU
S      M4.3, 1
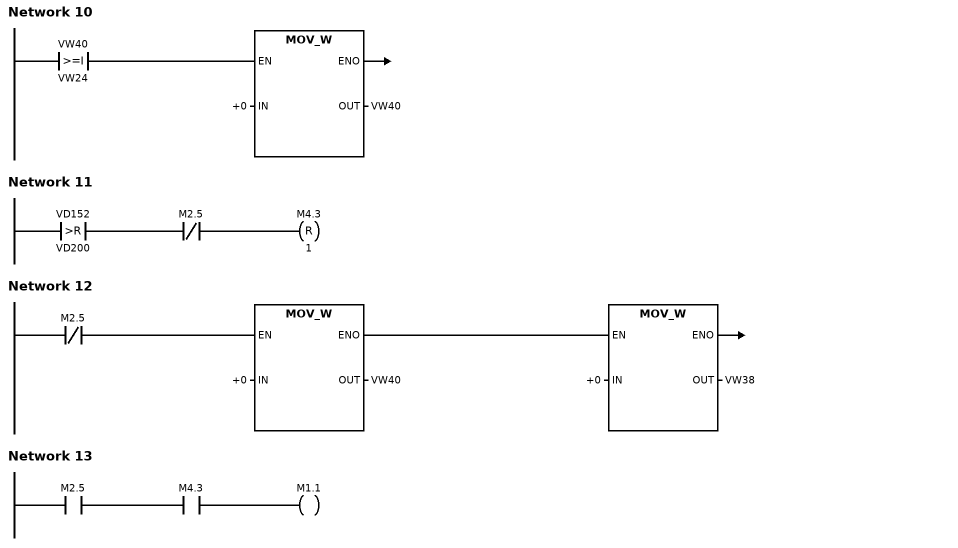
Network 10
LDW>=  VW40, VW24
MOVW   +0, VW40
Network 11
LDR>   VD152, VD200
AN     M2.5
R      M4.3, 1
Network 12
LDN    M2.5
MOVW   +0, VW40
AENO
MOVW   +0, VW38
Network 13
LD     M2.5
A      M4.3
=      M1.1
END_SUBROUTINE_BLOCK

SUBROUTINE_BLOCK VLT:SBR5
TITLE=
BEGIN
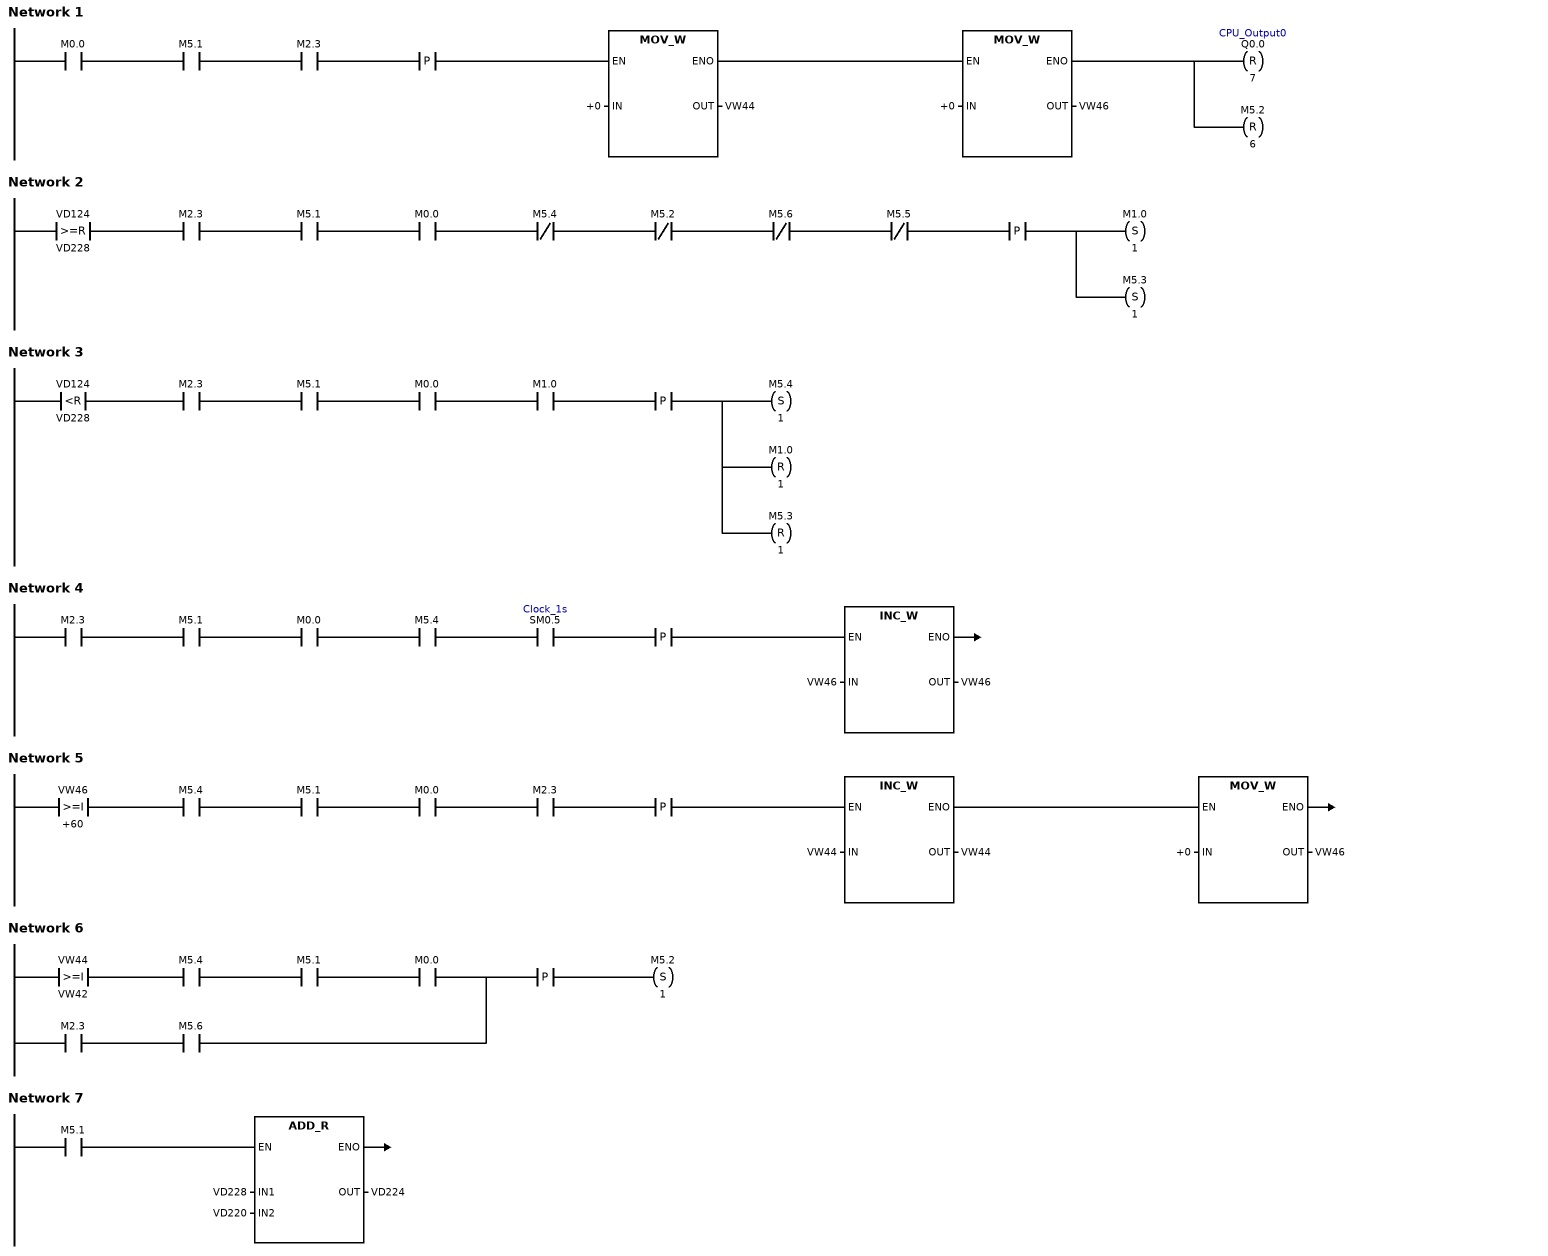
Network 1
LD     M0.0
A      M5.1
A      M2.3
EU
MOVW   +0, VW44
AENO
MOVW   +0, VW46
AENO
R      CPU_Output0:Q0.0, 7
R      M5.2, 6
Network 2
LDR>=  VD124, VD228
A      M2.3
A      M5.1
A      M0.0
AN     M5.4
AN     M5.2
AN     M5.6
AN     M5.5
EU
S      M1.0, 1
S      M5.3, 1
Network 3
LDR<   VD124, VD228
A      M2.3
A      M5.1
A      M0.0
A      M1.0
EU
S      M5.4, 1
R      M1.0, 1
R      M5.3, 1
Network 4
LD     M2.3
A      M5.1
A      M0.0
A      M5.4
A      Clock_1s:SM0.5
EU
INCW   VW46
Network 5
LDW>=  VW46, +60
A      M5.4
A      M5.1
A      M0.0
A      M2.3
EU
INCW   VW44
AENO
MOVW   +0, VW46
Network 6
LDW>=  VW44, VW42
A      M5.4
A      M5.1
A      M0.0
LD     M2.3
A      M5.6
OLD
EU
S      M5.2, 1
Network 7
LD     M5.1
MOVR   VD228, VD224
+R     VD220, VD224
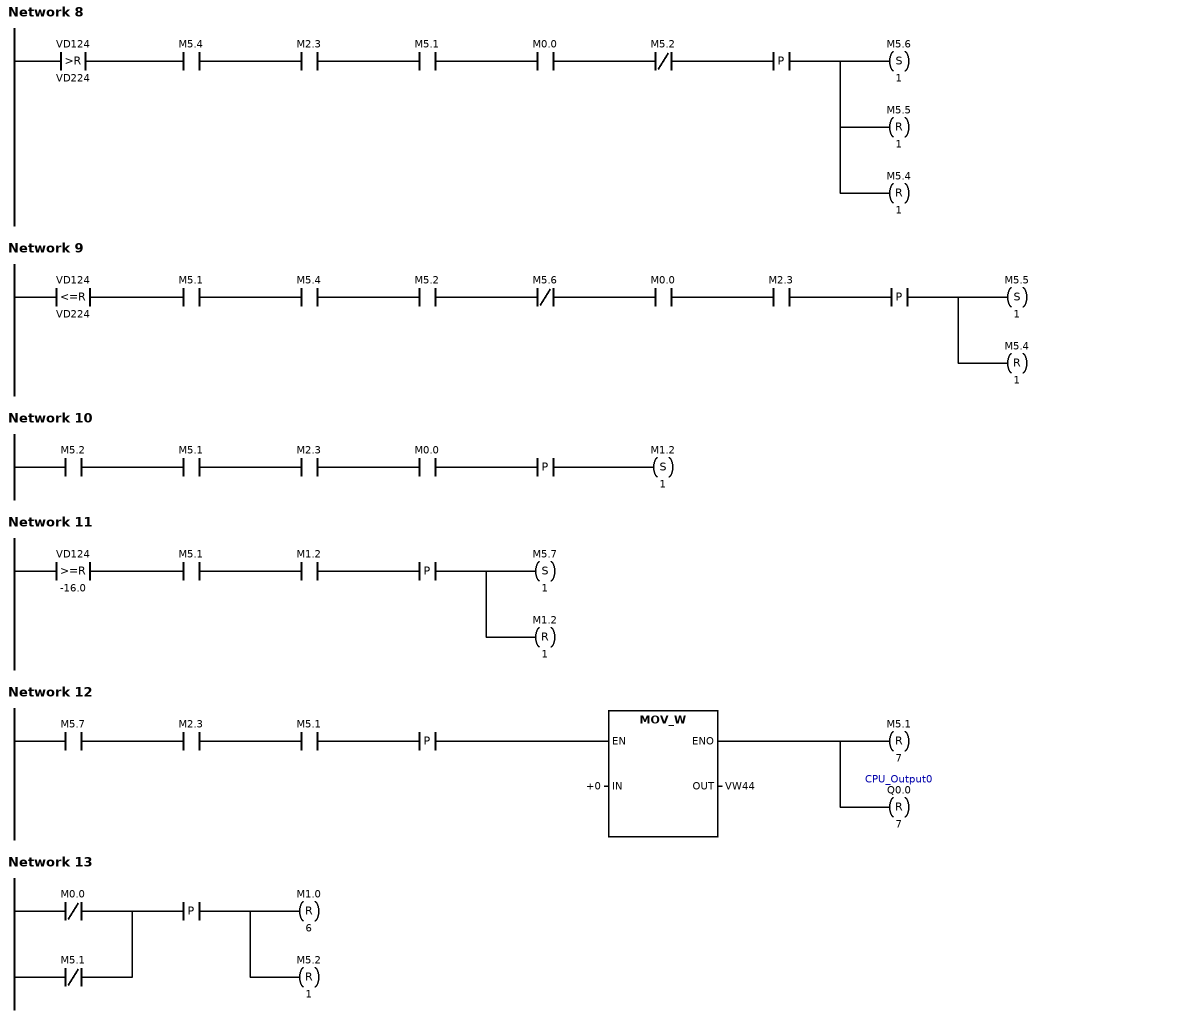
Network 8
LDR>   VD124, VD224
A      M5.4
A      M2.3
A      M5.1
A      M0.0
AN     M5.2
EU
S      M5.6, 1
R      M5.5, 1
R      M5.4, 1
Network 9
LDR<=  VD124, VD224
A      M5.1
A      M5.4
A      M5.2
AN     M5.6
A      M0.0
A      M2.3
EU
S      M5.5, 1
R      M5.4, 1
Network 10
LD     M5.2
A      M5.1
A      M2.3
A      M0.0
EU
S      M1.2, 1
Network 11
LDR>=  VD124, -16.0
A      M5.1
A      M1.2
EU
S      M5.7, 1
R      M1.2, 1
Network 12
LD     M5.7
A      M2.3
A      M5.1
EU
MOVW   +0, VW44
AENO
R      M5.1, 7
R      CPU_Output0:Q0.0, 7
Network 13
LDN    M0.0
ON     M5.1
EU
R      M1.0, 6
R      M5.2, 1
END_SUBROUTINE_BLOCK

// SBR6: protected block, not included

SUBROUTINE_BLOCK RTC:SBR7
TITLE=
BEGIN
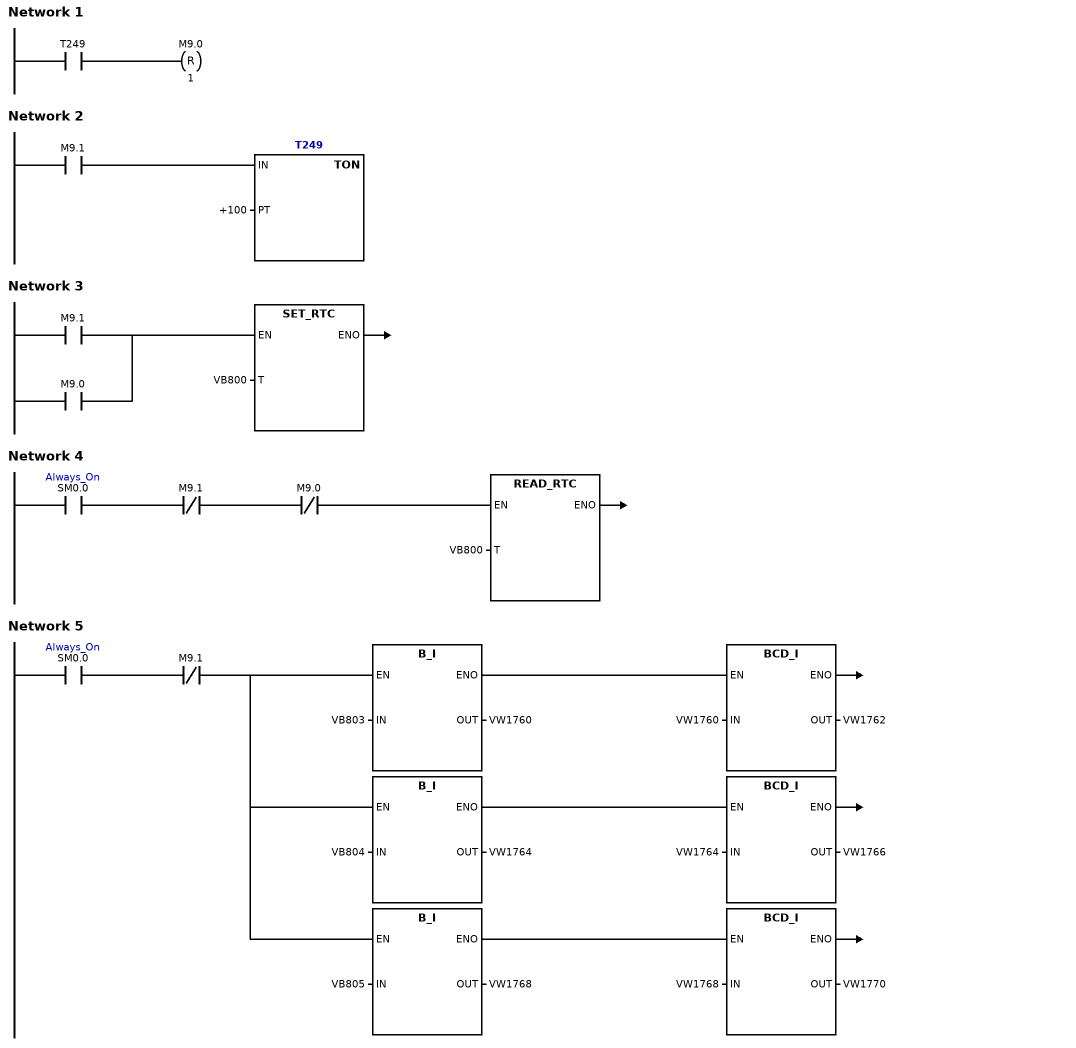
Network 1
LD     T249
R      M9.0, 1
Network 2
LD     M9.1
TON    T249, +100
Network 3
LD     M9.1
O      M9.0
TODW   VB800
Network 4
LD     Always_On:SM0.0
AN     M9.1
AN     M9.0
TODR   VB800
Network 5
LD     Always_On:SM0.0
AN     M9.1
LPS
BTI    VB803, VW1760
AENO
MOVW   VW1760, VW1762
BCDI   VW1762
LRD
BTI    VB804, VW1764
AENO
MOVW   VW1764, VW1766
BCDI   VW1766
LPP
BTI    VB805, VW1768
AENO
MOVW   VW1768, VW1770
BCDI   VW1770
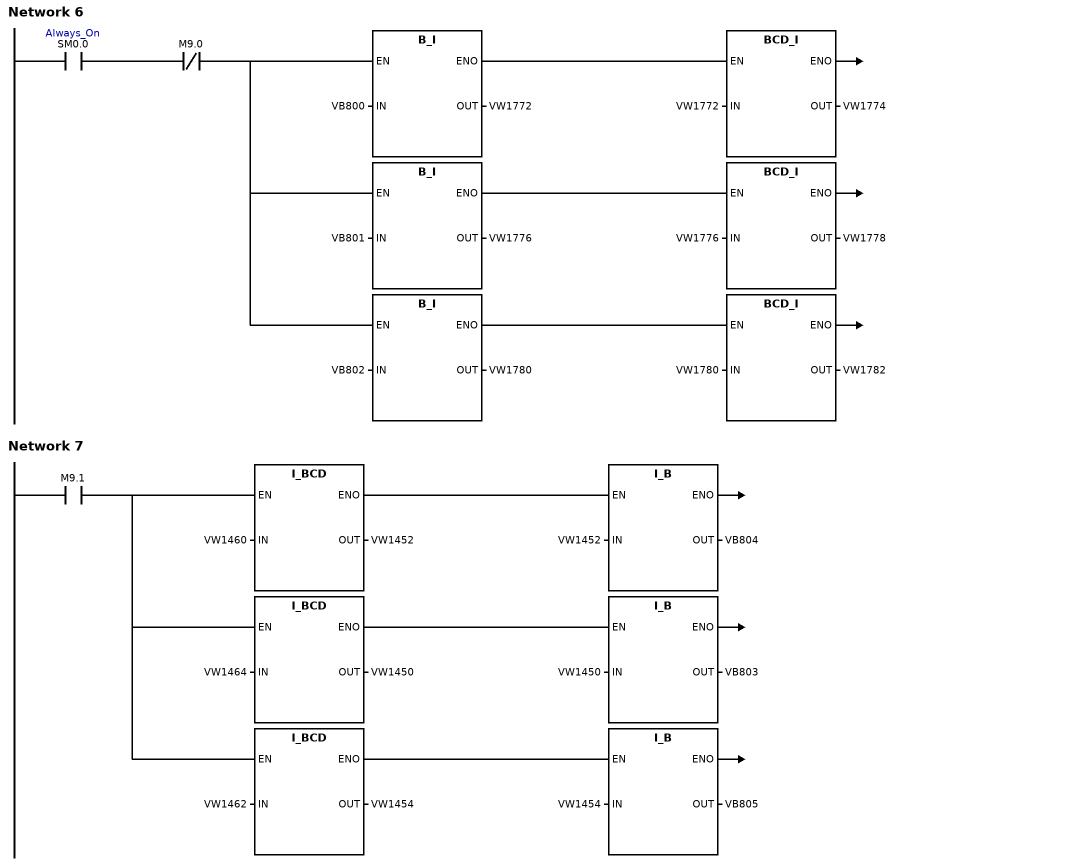
Network 6
LD     Always_On:SM0.0
AN     M9.0
LPS
BTI    VB800, VW1772
AENO
MOVW   VW1772, VW1774
BCDI   VW1774
LRD
BTI    VB801, VW1776
AENO
MOVW   VW1776, VW1778
BCDI   VW1778
LPP
BTI    VB802, VW1780
AENO
MOVW   VW1780, VW1782
BCDI   VW1782
Network 7
LD     M9.1
LPS
MOVW   VW1460, VW1452
AENO
IBCD   VW1452
AENO
ITB    VW1452, VB804
LRD
MOVW   VW1464, VW1450
AENO
IBCD   VW1450
AENO
ITB    VW1450, VB803
LPP
MOVW   VW1462, VW1454
AENO
IBCD   VW1454
AENO
ITB    VW1454, VB805
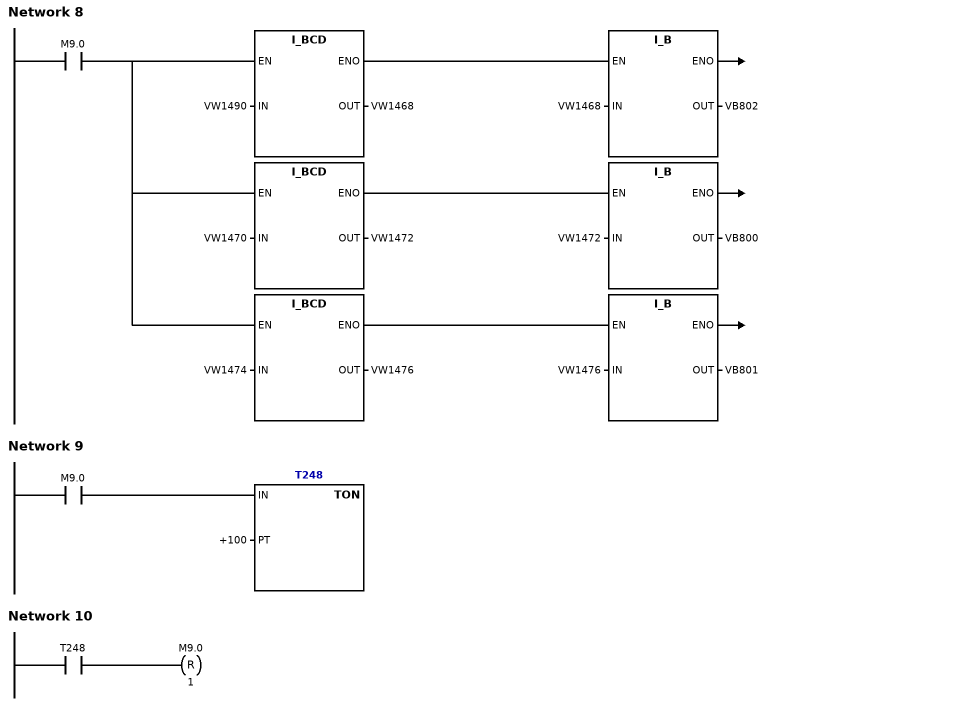
Network 8
LD     M9.0
LPS
MOVW   VW1490, VW1468
AENO
IBCD   VW1468
AENO
ITB    VW1468, VB802
LRD
MOVW   VW1470, VW1472
AENO
IBCD   VW1472
AENO
ITB    VW1472, VB800
LPP
MOVW   VW1474, VW1476
AENO
IBCD   VW1476
AENO
ITB    VW1476, VB801
Network 9
LD     M9.0
TON    T248, +100
Network 10
LD     T248
R      M9.0, 1
END_SUBROUTINE_BLOCK

SUBROUTINE_BLOCK Print:SBR8
TITLE=
BEGIN
